DATA_BLOCK "PilzData"   // DB2702
{ S7_Optimized_Access := 'FALSE' }
// stored: AutoNumber false
   VAR RETAIN
      "85A1" : Struct
         I8 : Bool;   // Light Current 1.1
         I9 : Bool;   // Light Current 1.2
         I10 : Bool;   // Light Current 2.1
         I11 : Bool;   // Light Current 2.2
         I12 : Bool;   // Stove E Stop_2.1
         I13 : Bool;   // Stove E Stop_2.2
         I14 : Bool;   // E Stop Feedback
         I15 : Bool;   // Safety Gate Feedback
         I0 : Bool;   // Control On
         I1 : Bool;   // Control Off
         I2 : Bool;   // Spare
         I3 : Bool;   // Spare
         I4 : Bool;   // E Stop_1.1
         I5 : Bool;   // E Stop_1.2
         I6 : Bool;   // Safety Gate 1.1
         I7 : Bool;   // Safety Gate 1.2
         I24 : Bool;
         I25 : Bool;
         I26 : Bool;
         I27 : Bool;
         I28 : Bool;
         I29 : Bool;
         I30 : Bool;
         I31 : Bool;
         I16 : Bool;   // Light Current 1 feedback
         I17 : Bool;   // Light Current 2 feedback
         I18 : Bool;   // Stove E Stop feedback
         I19 : Bool;   // Spare
         I20 : Bool;   // I20
         I21 : Bool;   // I21
         I22 : Bool;   // I22
         I23 : Bool;   // I23
         O0 : Bool;
         O1 : Bool;
         O2 : Bool;
         O3 : Bool;
         Spare_1 : Bool;
         Spare_2 : Bool;
         Spare_3 : Bool;
         Spare_4 : Bool;
         Spare_5 : Bool;
         Spare_6 : Bool;
         Spare_7 : Bool;
         Spare_8 : Bool;
         Spare_9 : Bool;
         Spare_10 : Bool;
         Spare_11 : Bool;
         Spare_12 : Bool;
      END_STRUCT;
      "85A2" : Struct
         I0 : Bool;   // UnLoadingMaterialDoor 1.1
         I1 : Bool;   // UnLoadingMaterialDoor 1.2
         I2 : Bool;   // UnLoadingMaterialDoor 2.1
         I3 : Bool;   // UnLoadingMaterialDoor 2.2
         I4 : Bool;   // UnLoadingMaterialDoor 3.1
         I5 : Bool;   // UnLoadingMaterialDoor 3.2
         I6 : Bool;   // LoadingMaterialDoor 4.1
         I7 : Bool;   // LoadingMaterialDoor 4.2
         O0 : Bool;
         O1 : Bool;
         O2 : Bool;
         O3 : Bool;
         Spare_1 : Bool;
         Spare_2 : Bool;
         Spare_3 : Bool;
         Spare_4 : Bool;
      END_STRUCT;
      "85A3" : Struct
         I0 : Bool;   // MaterialDoor 1 feedback
         I1 : Bool;   // MaterialDoor 2 feedback
         I2 : Bool;   // MaterialDoor 3 feedback
         I3 : Bool;   // MaterialDoor 4 feedback
         I4 : Bool;   // Stove Door feedback 1.1
         I5 : Bool;   // Stove Door feedback 1.2
         I6 : Bool;   // Robot feedback
         I7 : Bool;   // Robot Door feedback
         O0 : Bool;
         O1 : Bool;
         O2 : Bool;
         O3 : Bool;
         Spare_1 : Bool;
         Spare_2 : Bool;
         Spare_3 : Bool;
         Spare_4 : Bool;
      END_STRUCT;
      "85A4" : Struct
         I0 : Bool;   // LoadingMaterialDoor 1.1
         I1 : Bool;   // LoadingMaterialDoor 1.2
         I2 : Bool;   // LoadingMaterialDoor 2.1
         I3 : Bool;   // LoadingMaterialDoor 2.2
         I4 : Bool;   // LoadingMaterialDoor 3.1
         I5 : Bool;   // LoadingMaterialDoor 3.2
         I6 : Bool;   // NG 2 Door 1.1
         I7 : Bool;   // NG 2 Door 1.2
         O0 : Bool;
         O1 : Bool;
         O2 : Bool;
         O3 : Bool;
         Spare_1 : Bool;
         Spare_2 : Bool;
         Spare_3 : Bool;
         Spare_4 : Bool;
      END_STRUCT;
      "85A5" : Struct
         I0 : Bool;   // Robot 1 E Stop1.1
         I1 : Bool;   // Robot 1 E Stop1.2
         I2 : Bool;   // Robot 2 E Stop1.1
         I3 : Bool;   // Robot 2 E Stop1.2
         I4 : Bool;   // Robot 3 E Stop1.1
         I5 : Bool;   // Robot 3 E Stop1.2
         I6 : Bool;   // NG 1 Door 1.1
         I7 : Bool;   // NG 1 Door 1.2
         O0 : Bool;
         O1 : Bool;
         O2 : Bool;
         O3 : Bool;
         Spare_1 : Bool;
         Spare_2 : Bool;
         Spare_3 : Bool;
         Spare_4 : Bool;
      END_STRUCT;
      TON { S7_SetPoint := 'True'} : Array[0..50] of TON_TIME;
      OK_BoxFlag : Struct
         X_Moving : Bool;
         Y_Pulling : Bool;
         X_Need_MoveBox : Bool;
         Y_Need_PullBox : Bool;
         Pushing : Bool;
         ChangeUnloadingBox : Bool;
         HMIChangeUnloadingBox : Bool;
         ManualOKBox : Bool;
         HMIManualOKBox : Int;
      END_STRUCT;
      Status : Int;
   END_VAR
BEGIN
END_DATA_BLOCK

DATA_BLOCK "GluingControl"   // DB2800
{ S7_Optimized_Access := 'FALSE' }
// stored: AutoNumber false
   VAR
      Input : Struct
         GluingDeviceReady : Bool;
         GluingFault : Bool;
         GluingRefillTank : Bool;
         GluingTankEmpty : Bool;
      END_STRUCT;
      Output : Struct
         GluingPro_X : Bool;
         GluingPro_Y : Bool;
         GluingPro_Z : Bool;
         GluingReset : Bool;
      END_STRUCT;
      Control : Struct
         Manual_X : Bool;
         Manual_Y : Bool;
         Manual_Z : Bool;
         Manual_Control : Int;
         Auto_Start : Bool;
         Auto_Y : Bool;
         Auto_Z : Bool;
         Auto_Control : Int;
         ManualTest_X : Bool;
         ManualTestStartGlue : Bool;
      END_STRUCT;
      GlueCalibratonMode : Bool;
      TON : Array[1..10] of IEC_LTIMER;
      P { S7_SetPoint := 'True'} : Array[1..10] of Bool;
      GlueInitiaStart : Bool;
   END_VAR
BEGIN
END_DATA_BLOCK

DATA_BLOCK "PalletNGData"   // DB2900
{ S7_Optimized_Access := 'FALSE' }
// stored: AutoNumber false
   VAR
      LoadingNGPallet : Struct
         NG_1_1 : Bool;
         NG_1_2 : Bool;
         NG_1_3 : Bool;
         NG_1_4 : Bool;
         NG_1_5 : Bool;
         NG_2_1 : Bool;
         NG_2_2 : Bool;
         NG_2_3 : Bool;
         NG_2_4 : Bool;
         NG_2_5 : Bool;
         NG_3_1 : Bool;
         NG_3_2 : Bool;
         NG_3_3 : Bool;
         NG_3_4 : Bool;
         NG_3_5 : Bool;
         OpenFlag : Bool;
         Status_1 : Int;
         Status_2 : Int;
         Status_3 : Int;
         Ready_1 : Bool;
         Ready_2 : Bool;
         Ready_3 : Bool;
         Ready_4 : Bool;
         Ready_5 : Bool;
         Ready_6 : Bool;
         Ready : Bool;
         Interlock_1 : Array[1..10] of Bool;
         Interlock_2 : Array[1..10] of Bool;
         Interlock_3 : Array[1..10] of Bool;
         LockStatus : Int;
      END_STRUCT;
      UnLoadingNGPallet : Struct
         NG_1_1 : Bool;
         NG_1_2 : Bool;
         NG_1_3 : Bool;
         NG_1_4 : Bool;
         NG_1_5 : Bool;
         NG_2_1 : Bool;
         NG_2_2 : Bool;
         NG_2_3 : Bool;
         NG_2_4 : Bool;
         NG_2_5 : Bool;
         NG_3_1 : Bool;
         NG_3_2 : Bool;
         NG_3_3 : Bool;
         NG_3_4 : Bool;
         NG_3_5 : Bool;
         OpenFlag : Bool;
         Status_1 : Int;
         Status_2 : Int;
         Status_3 : Int;
         Ready_1 : Bool;
         Ready_2 : Bool;
         Ready_3 : Bool;
         Ready_4 : Bool;
         Ready_5 : Bool;
         Ready_6 : Bool;
         Ready : Bool;
         Interlock_1 : Array[1..10] of Bool;
         Interlock_2 : Array[1..10] of Bool;
         Interlock_3 : Array[1..10] of Bool;
         LockStatus : Int;
      END_STRUCT;
      P : Array[0..10] of Bool;
   END_VAR
BEGIN
END_DATA_BLOCK

DATA_BLOCK "MotorControl"   // DB3100
{ S7_Optimized_Access := 'TRUE' }
// stored: AutoNumber false, MemoryReserve 100
   VAR
      Dev : Array[1..20] of "Motor_Control";
   END_VAR
BEGIN
END_DATA_BLOCK

DATA_BLOCK "MotorData"   // DB3120
{ S7_Optimized_Access := 'FALSE' }
// stored: AutoNumber false
   VAR
      Ton : Array[0..50] of TON_TIME;
      P { S7_SetPoint := 'True'} : Array[0..50] of Bool;
      "Time" : Array[0..50] of Time;
   END_VAR
BEGIN
   "Time"[0..50] := T#60s;
END_DATA_BLOCK

DATA_BLOCK "KistlerPressData1"   // DB2311
{ S7_Optimized_Access := 'FALSE' }
// stored: AutoNumber false
   VAR
      Spare : Struct
         Spare : Array[0..85] of Byte;
      END_STRUCT;
      Data : Struct
         EO01 : Struct
            "pvXMin-Y" : Real;
            "pvXMax-Y" : Real;
            "pvXMin-X" : Real;
            "pvXMax-X" : Real;
         END_STRUCT;
         EO02 : Struct
            "pvXMin-Y" : Real;
            "pvXMax-Y" : Real;
            "pvXMin-X" : Real;
            "pvXMax-X" : Real;
         END_STRUCT;
         EO03 : Struct
            "pvXMax-Y" : Real;
            "pvXMax-X" : Real;
         END_STRUCT;
      END_STRUCT;
      iWritePressData : Struct
         temp1 : Real;
      END_STRUCT;
      PressData1 : Struct
         pvBlock_X : Real;
         pvBlock_Y : Real;
      END_STRUCT;
      PressData2 : Struct
         pvBlock_X : Real;
         pvBlock_Y : Real;
      END_STRUCT;
      ManualPro : Int;
   END_VAR
BEGIN
END_DATA_BLOCK

DATA_BLOCK "KistlerPresser1_DB"   // DB2312
{ S7_Optimized_Access := 'FALSE' }
// stored: AutoNumber false
   VAR
      ShaftID : Array[0..50] of Char;
      HousingID_1 : Array[0..50] of Char;
      HousingID_2 : Array[0..50] of Char;
      Shaft : String[48];
      spare : String[48] := '46';
   END_VAR
BEGIN
END_DATA_BLOCK

DATA_BLOCK "KistlerPressData2"   // DB2321
{ S7_Optimized_Access := 'FALSE' }
// stored: AutoNumber false
   VAR
      Spare : Struct
         Spare : Array[0..85] of Byte;
      END_STRUCT;
      Data : Struct
         EO01 : Struct
            "pvXMin-Y" : Real;
            "pvXMax-Y" : Real;
            "pvXMin-X" : Real;
            "pvXMax-X" : Real;
         END_STRUCT;
         EO02 : Struct
            "pvXMin-Y" : Real;
            "pvXMax-Y" : Real;
            "pvXMin-X" : Real;
            "pvXMax-X" : Real;
         END_STRUCT;
         EO03 : Struct
            "pvXMax-Y" : Real;
            "pvXMax-X" : Real;
         END_STRUCT;
      END_STRUCT;
      iWritePressData : Struct
         temp1 : Real;
      END_STRUCT;
      PressData1 : Struct
         pvBlock_X : Real;
         pvBlock_Y : Real;
      END_STRUCT;
      ManualPro : Int;
   END_VAR
BEGIN
END_DATA_BLOCK

DATA_BLOCK "KistlerPresser2_DB"   // DB2322
{ S7_Optimized_Access := 'FALSE' }
// stored: AutoNumber false
   VAR
      ShaftID : Array[0..50] of Char;
      HousingID_1 : Array[0..50] of Char;
      HousingID_2 : Array[0..50] of Char;
      Shaft : String[48];
      spare : String[48] := '46';
   END_VAR
BEGIN
END_DATA_BLOCK

DATA_BLOCK "ST10_FB_Tower_4Lamp_DB"
{ S7_Optimized_Access := 'TRUE' }
VERSION : 0.1
NON_RETAIN
// ATTRIBUTES
// AUTO_NUMBER = False
// BLOCK_NUMBER = 5050
// END_ATTRIBUTES
"FB_Tower_4Lamp"

BEGIN

END_DATA_BLOCK

DATA_BLOCK "DB_ProcessSlots"
{ S7_Optimized_Access := 'TRUE' }
VERSION : 0.1
// ATTRIBUTES
// AUTO_NUMBER = False
// BLOCK_NUMBER = 2600
// END_ATTRIBUTES
   VAR 
      Slots : Array[1..16] of "UDT_ProcessSlot";
   END_VAR


BEGIN
   Slots[1].SlotID := 1;
   Slots[1].PositionTag := 'A_ScanRotate';
   Slots[2].SlotID := 2;
   Slots[2].PositionTag := 'F_Robot1Grip1';
   Slots[3].SlotID := 3;
   Slots[3].PositionTag := 'F_Robot1Grip2';
   Slots[4].SlotID := 4;
   Slots[4].PositionTag := 'B_Press1';
   Slots[5].SlotID := 5;
   Slots[5].PositionTag := 'C_Glue';
   Slots[6].SlotID := 6;
   Slots[6].PositionTag := 'F_Robot2Grip1';
   Slots[7].SlotID := 7;
   Slots[7].PositionTag := 'F_Robot2Grip2';
   Slots[8].SlotID := 8;
   Slots[8].PositionTag := 'C_GlueNGBuffer';
   Slots[9].SlotID := 9;
   Slots[9].PositionTag := 'C_MagnScanNGBuffer';
   Slots[10].SlotID := 10;
   Slots[10].PositionTag := 'B_Press2';
   Slots[11].SlotID := 11;
   Slots[11].PositionTag := 'F_Robot3Grip1';
   Slots[12].SlotID := 12;
   Slots[12].PositionTag := 'F_Robot3Grip2';
   Slots[13].SlotID := 13;
   Slots[13].PositionTag := 'H_ShafeLine';
   Slots[14].SlotID := 14;
   Slots[14].PositionTag := 'J_ShafeLine';
   Slots[15].SlotID := 15;
   Slots[15].PositionTag := 'K_ShafeLine';
   Slots[16].SlotID := 16;
   Slots[16].PositionTag := 'L_ShafeLine';

END_DATA_BLOCK

DATA_BLOCK "DB_ProcessSlots_Global"
{ S7_Optimized_Access := 'TRUE' }
VERSION : 0.1
// ATTRIBUTES
// AUTO_NUMBER = False
// BLOCK_NUMBER = 2601
// END_ATTRIBUTES
   VAR 
      SlotHasProduct : Array[1..16] of Bool;
      SlotLocked : Array[1..16] of Bool;
      SlotPendingWrite : Array[1..16] of Bool;
      ActiveRecipeID : Int;
      ActiveRecipeVersion : String[18];
      BufferIndex : Int;
   END_VAR


BEGIN
   ActiveRecipeID := 1;
   ActiveRecipeVersion := 'INIT';
   BufferIndex := 1;

END_DATA_BLOCK

DATA_BLOCK "DB_RecipeActiveNew"
{ S7_Optimized_Access := 'TRUE' }
VERSION : 0.1
// ATTRIBUTES
// AUTO_NUMBER = False
// BLOCK_NUMBER = 2701
// END_ATTRIBUTES
   VAR 
      Header : "UDT_RecipeHeader";
      SubProcess : Array[1..16] of "UDT_SubProcessRecipe";
      FixtureCodes : Array[1..16] of String[128];
      GripperCodes : Array[1..12] of String[128];
      PressPrograms : Array[1..4] of Int;
      VisionPrograms : Array[1..8] of Int;
   END_VAR


BEGIN
   Header.ProductName := 'ACTIVE';
   Header.ProductID := 'ACTIVE';
   Header.RecipeVersion := 'PENDING';
   Header.Enabled := FALSE;

END_DATA_BLOCK

DATA_BLOCK "DB_RecipeMaster"
{ S7_Optimized_Access := 'TRUE' }
VERSION : 0.1
// ATTRIBUTES
// AUTO_NUMBER = False
// BLOCK_NUMBER = 2700
// END_ATTRIBUTES
   VAR 
      Header : "UDT_RecipeHeader";
      SubProcess : Array[1..32] of "UDT_SubProcessRecipe";
      FixtureCodes : Array[1..16] of String[128];
      GripperCodes : Array[1..18] of String[128];
      VisionPrograms : Array[1..16] of Int;
   END_VAR


BEGIN
   Header.ProductName := 'Product_1';
   Header.ProductID := 'P1';
   Header.RecipeVersion := 'V1.0';
   Header.FixtureFamily := 1;
   Header.Enabled := TRUE;
   Header.CreatedBy := 'OP10';
   Header.UpdatedBy := 'OP10';
   Header.Comment := 'Seed recipe migrated from ST10_RecipeDB';

   FixtureCodes[1] := 'SZ23055-OP010-E-Compressor-ring1 Loading tooling-1';
   FixtureCodes[2] := 'SZ23055-OP010-E-Compressor-ring1 Loading tooling-2';
   FixtureCodes[3] := 'SZ23055-OP010-E-Compressor-ring1 Loading tooling-3';
   FixtureCodes[4] := 'SZ23055-OP010-E-Compressor-ring1 Loading tooling-4';
   FixtureCodes[5] := 'SZ23055-OP010-E-Compressor-ring1 Loading tooling-5';
   FixtureCodes[6] := 'SZ23055-OP010-E-Compressor-ring1 Loading tooling-6';
   FixtureCodes[7] := 'SZ23055-OP010-E-Compressor-ring1 Loading tooling-7';
   FixtureCodes[8] := 'SZ23055-OP010-E-Compressor-ring1 Loading tooling-8';
   FixtureCodes[9] := 'SZ23055-OP010-E-Compressor-ring2 Loading tooling-1';
   FixtureCodes[10] := 'SZ23055-OP010-E-Compressor-ring2 Loading tooling-2';
   FixtureCodes[11] := 'SZ23055-OP010-E-Compressor-ring2 Loading tooling-3';
   FixtureCodes[12] := 'SZ23055-OP010-E-Compressor-ring2 Loading tooling-4';

   GripperCodes[1] := 'SZ23055-OP010-E-Compressor-robot1 ring1 Left clamping jaw tooling-1';
   GripperCodes[2] := 'SZ23055-OP010-E-Compressor-robot1 ring1 Right clamping jaw tooling-2';
   GripperCodes[3] := 'SZ23055-OP010-E-Compressor-robot1 shaft Left clamping jaw tooling-1';
   GripperCodes[4] := 'SZ23055-OP010-E-Compressor-robot1 shaft Right clamping jaw tooling-2';
   GripperCodes[5] := 'SZ23055-OP010-E-Compressor-robot2 shaft Right clamping jaw tooling-2';
   GripperCodes[6] := 'SZ23055-OP010-E-Compressor-robot2 shaft Left clamping jaw tooling-1';

END_DATA_BLOCK

DATA_BLOCK "ST10_CountCycleTimeMain_DB"
{ S7_Optimized_Access := 'TRUE' }
VERSION : 0.1
NON_RETAIN
// ATTRIBUTES
// AUTO_NUMBER = False
// BLOCK_NUMBER = 1009
// END_ATTRIBUTES
"ST10_CountCycleTimeMain"

BEGIN

END_DATA_BLOCK

DATA_BLOCK "DB_MESLoadData"
{ S7_Optimized_Access := 'TRUE' }
VERSION : 0.1
// ATTRIBUTES
// AUTO_NUMBER = False
// BLOCK_NUMBER = 2800
// END_ATTRIBUTES
   VAR 
      Station1 : "UDT_MESLoadData";
      Station2 : "UDT_MESLoadData";
      Station3 : "UDT_MESLoadData";
      Station4 : "UDT_MESLoadData";
   END_VAR


BEGIN

END_DATA_BLOCK

DATA_BLOCK "DT-Chars_DB"
{ S7_Optimized_Access := 'FALSE' }
VERSION : 0.1
NON_RETAIN
// ATTRIBUTES
// AUTO_NUMBER = False
// BLOCK_NUMBER = 2360
// END_ATTRIBUTES
"DT-Chars"

BEGIN

END_DATA_BLOCK

DATA_BLOCK "MES_CHeck_DB"
{ S7_Optimized_Access := 'TRUE' }
VERSION : 0.1
NON_RETAIN
// ATTRIBUTES
// AUTO_NUMBER = False
// BLOCK_NUMBER = 111
// END_ATTRIBUTES
"MES_CHeck"

BEGIN

END_DATA_BLOCK

DATA_BLOCK "PartDataManage_Part1_DB"
{ S7_Optimized_Access := 'TRUE' }
VERSION : 0.1
NON_RETAIN
// ATTRIBUTES
// AUTO_NUMBER = True
// BLOCK_NUMBER = 1501
// END_ATTRIBUTES
"PartDataManage"

BEGIN

END_DATA_BLOCK

DATA_BLOCK "PartDataManage_Part2_DB"
{ S7_Optimized_Access := 'TRUE' }
VERSION : 0.1
NON_RETAIN
"PartDataManage"

BEGIN

END_DATA_BLOCK

DATA_BLOCK "PartDataManage_Part3_DB"
{ S7_Optimized_Access := 'TRUE' }
VERSION : 0.1
NON_RETAIN
// ATTRIBUTES
// AUTO_NUMBER = True
// BLOCK_NUMBER = 1503
// END_ATTRIBUTES
"PartDataManage"

BEGIN

END_DATA_BLOCK

DATA_BLOCK "PartDataManage_Part4_DB"
{ S7_Optimized_Access := 'TRUE' }
VERSION : 0.1
NON_RETAIN
// ATTRIBUTES
// AUTO_NUMBER = True
// BLOCK_NUMBER = 1504
// END_ATTRIBUTES
"PartDataManage"

BEGIN

END_DATA_BLOCK

DATA_BLOCK "MB_CLIENT_DB"
{InstructionName := 'MB_CLIENT';
 LibVersion := '5.1';
 S7_Optimized_Access := 'TRUE' }
AUTHOR : SIMATIC
FAMILY : MBUS_TCP
NAME : MB_CLI
VERSION : 5.1
NON_RETAIN
MB_CLIENT

BEGIN

END_DATA_BLOCK

DATA_BLOCK "ST10_SystemModeFB_iDB"
{ S7_Optimized_Access := 'TRUE' }
VERSION : 0.1
NON_RETAIN
// ATTRIBUTES
// AUTO_NUMBER = False
// BLOCK_NUMBER = 1000
// END_ATTRIBUTES
"SystemMode"

BEGIN

END_DATA_BLOCK

DATA_BLOCK "AutoProcessDataPopUp_DB"
{ S7_Optimized_Access := 'TRUE' }
VERSION : 0.1
NON_RETAIN
// ATTRIBUTES
// AUTO_NUMBER = True
// BLOCK_NUMBER = 2
// END_ATTRIBUTES
"AutoProcessDataPopUp"

BEGIN

END_DATA_BLOCK

DATA_BLOCK "ST10_Flow11_A2TableScan_iDB"
{ S7_Optimized_Access := 'TRUE' }
VERSION : 0.1
NON_RETAIN
// ATTRIBUTES
// AUTO_NUMBER = False
// BLOCK_NUMBER = 1081
// END_ATTRIBUTES
"ST10_Flow11_A2TableScan"

BEGIN

END_DATA_BLOCK

DATA_BLOCK "ST10_Flow12_A2TableUnloading_iDB"
{ S7_Optimized_Access := 'TRUE' }
VERSION : 0.1
NON_RETAIN
// ATTRIBUTES
// AUTO_NUMBER = False
// BLOCK_NUMBER = 1082
// END_ATTRIBUTES
"ST10_Flow12_A2TableUnloading"

BEGIN

END_DATA_BLOCK

DATA_BLOCK "ST10_Flow14_B2Press_iDB"
{ S7_Optimized_Access := 'TRUE' }
VERSION : 0.1
NON_RETAIN
// ATTRIBUTES
// AUTO_NUMBER = False
// BLOCK_NUMBER = 1084
// END_ATTRIBUTES
"ST10_Flow14_B2Press"

BEGIN

END_DATA_BLOCK

DATA_BLOCK "ST10_Flow15_FRobot_3_iDB"
{ S7_Optimized_Access := 'TRUE' }
VERSION : 0.1
NON_RETAIN
// ATTRIBUTES
// AUTO_NUMBER = False
// BLOCK_NUMBER = 1085
// END_ATTRIBUTES
"ST10_Flow15_FRobot_3"

BEGIN

END_DATA_BLOCK

DATA_BLOCK "ST10_Flow1_A1TableScan_iDB"
{ S7_Optimized_Access := 'TRUE' }
VERSION : 0.1
NON_RETAIN
"ST10_Flow1_A1TableScan"

BEGIN

END_DATA_BLOCK

DATA_BLOCK "ST10_Flow21_HShaftLifting_iDB"
{ S7_Optimized_Access := 'TRUE' }
VERSION : 0.1
NON_RETAIN
// ATTRIBUTES
// AUTO_NUMBER = False
// BLOCK_NUMBER = 1091
// END_ATTRIBUTES
"ST10_Flow21_HShaftLifting"

BEGIN

END_DATA_BLOCK

DATA_BLOCK "ST10_Flow22_JMagnetLifting_iDB"
{ S7_Optimized_Access := 'TRUE' }
VERSION : 0.1
NON_RETAIN
"ST10_Flow22_JMagnetLifting"

BEGIN

END_DATA_BLOCK

DATA_BLOCK "ST10_Flow23_KReserveLifting_iDB"
{ S7_Optimized_Access := 'TRUE' }
VERSION : 0.1
NON_RETAIN
// ATTRIBUTES
// AUTO_NUMBER = False
// BLOCK_NUMBER = 1093
// END_ATTRIBUTES
"ST10_Flow23_KReserveLifting"

BEGIN

END_DATA_BLOCK

DATA_BLOCK "ST10_Flow24_LUnloadingTrans_iDB"
{ S7_Optimized_Access := 'TRUE' }
VERSION : 0.1
NON_RETAIN
// ATTRIBUTES
// AUTO_NUMBER = False
// BLOCK_NUMBER = 1094
// END_ATTRIBUTES
"ST10_Flow24_LUnloadingTrans"

BEGIN

END_DATA_BLOCK

DATA_BLOCK "ST10_Flow25_HShaftLoad&Unload_iDB"
{ S7_Optimized_Access := 'TRUE' }
VERSION : 0.1
NON_RETAIN
// ATTRIBUTES
// AUTO_NUMBER = False
// BLOCK_NUMBER = 1095
// END_ATTRIBUTES
"ST10_Flow25_HShaftLoad&Unload"

BEGIN

END_DATA_BLOCK

DATA_BLOCK "ST10_Flow26_JMagnetLoad&Unload_iDB"
{ S7_Optimized_Access := 'TRUE' }
VERSION : 0.1
NON_RETAIN
// ATTRIBUTES
// AUTO_NUMBER = False
// BLOCK_NUMBER = 1096
// END_ATTRIBUTES
"ST10_Flow26_JMagnetLoad&Unload"

BEGIN

END_DATA_BLOCK

DATA_BLOCK "ST10_Flow27_KReserveLoad&Unload_iDB"
{ S7_Optimized_Access := 'TRUE' }
VERSION : 0.1
NON_RETAIN
// ATTRIBUTES
// AUTO_NUMBER = False
// BLOCK_NUMBER = 1097
// END_ATTRIBUTES
"ST10_Flow27_KReserveLoad&Unload"

BEGIN

END_DATA_BLOCK

DATA_BLOCK "ST10_Flow28_LUnloadingLoad&Unload_IiDB"
{ S7_Optimized_Access := 'TRUE' }
VERSION : 0.1
NON_RETAIN
"ST10_Flow28_LUnloadingLoad&Unload"

BEGIN

END_DATA_BLOCK

DATA_BLOCK "ST10_Flow2_A1TableUnloading_iDB"
{ S7_Optimized_Access := 'TRUE' }
VERSION : 0.1
NON_RETAIN
"ST10_Flow2_A1TableUnloading"

BEGIN

END_DATA_BLOCK

DATA_BLOCK "ST10_Flow3_A1RotaryScan_iDB"
{ S7_Optimized_Access := 'TRUE' }
VERSION : 0.1
NON_RETAIN
// ATTRIBUTES
// AUTO_NUMBER = False
// BLOCK_NUMBER = 1073
// END_ATTRIBUTES
"ST10_Flow3_A1RotaryShaftScan"

BEGIN

END_DATA_BLOCK

DATA_BLOCK "ST10_Flow4_B1Press_iDB"
{ S7_Optimized_Access := 'TRUE' }
VERSION : 0.1
NON_RETAIN
"ST10_Flow4_B1Press"

BEGIN

END_DATA_BLOCK

DATA_BLOCK "ST10_Flow5_FRobot_1_iDB"
{ S7_Optimized_Access := 'TRUE' }
VERSION : 0.1
NON_RETAIN
"ST10_Flow5_FRobot_1"

BEGIN

END_DATA_BLOCK

DATA_BLOCK "ST10_Flow6_FixtureCodeScan_iDB"
{ S7_Optimized_Access := 'TRUE' }
VERSION : 0.1
NON_RETAIN
"ST10_Flow6_ToolCodeScan"

BEGIN

END_DATA_BLOCK

DATA_BLOCK "ST10_Flow7_CGlueing_iDB"
{ S7_Optimized_Access := 'TRUE' }
VERSION : 0.1
NON_RETAIN
"ST10_Flow7_CGlueing"

BEGIN

END_DATA_BLOCK

DATA_BLOCK "ST10_Flow8_FRobot_2_iDB"
{ S7_Optimized_Access := 'TRUE' }
VERSION : 0.1
NON_RETAIN
// ATTRIBUTES
// AUTO_NUMBER = False
// BLOCK_NUMBER = 1078
// END_ATTRIBUTES
"ST10_Flow8_FRobot_2"

BEGIN

END_DATA_BLOCK

DATA_BLOCK "ST10_MaterialGate1_DB"
{ S7_Optimized_Access := 'FALSE' }
VERSION : 0.1
NON_RETAIN
// ATTRIBUTES
// AUTO_NUMBER = False
// BLOCK_NUMBER = 1151
// END_ATTRIBUTES
"SafetyGate"

BEGIN

END_DATA_BLOCK

DATA_BLOCK "ST10_MaterialGate2_DB"
{ S7_Optimized_Access := 'FALSE' }
VERSION : 0.1
NON_RETAIN
// ATTRIBUTES
// AUTO_NUMBER = False
// BLOCK_NUMBER = 1152
// END_ATTRIBUTES
"SafetyGate"

BEGIN

END_DATA_BLOCK

DATA_BLOCK "ST10_MaterialGate3_DB"
{ S7_Optimized_Access := 'FALSE' }
VERSION : 0.1
NON_RETAIN
// ATTRIBUTES
// AUTO_NUMBER = False
// BLOCK_NUMBER = 1153
// END_ATTRIBUTES
"SafetyGate"

BEGIN

END_DATA_BLOCK

DATA_BLOCK "ST10_MaterialGate4_DB"
{ S7_Optimized_Access := 'FALSE' }
VERSION : 0.1
NON_RETAIN
// ATTRIBUTES
// AUTO_NUMBER = False
// BLOCK_NUMBER = 1154
// END_ATTRIBUTES
"SafetyGate"

BEGIN

END_DATA_BLOCK

DATA_BLOCK "ST10_MaterialGate5_DB"
{ S7_Optimized_Access := 'FALSE' }
VERSION : 0.1
NON_RETAIN
// ATTRIBUTES
// AUTO_NUMBER = False
// BLOCK_NUMBER = 1155
// END_ATTRIBUTES
"SafetyGate"

BEGIN

END_DATA_BLOCK

DATA_BLOCK "ST10_MaterialGate6_DB"
{ S7_Optimized_Access := 'FALSE' }
VERSION : 0.1
NON_RETAIN
// ATTRIBUTES
// AUTO_NUMBER = False
// BLOCK_NUMBER = 1156
// END_ATTRIBUTES
"SafetyGate"

BEGIN

END_DATA_BLOCK

DATA_BLOCK "ST10_MaterialGate7_DB"
{ S7_Optimized_Access := 'FALSE' }
VERSION : 0.1
NON_RETAIN
// ATTRIBUTES
// AUTO_NUMBER = False
// BLOCK_NUMBER = 1157
// END_ATTRIBUTES
"SafetyGate"

BEGIN

END_DATA_BLOCK

DATA_BLOCK "ST10_NGGate1_DB"
{ S7_Optimized_Access := 'FALSE' }
VERSION : 0.1
NON_RETAIN
// ATTRIBUTES
// AUTO_NUMBER = False
// BLOCK_NUMBER = 1158
// END_ATTRIBUTES
"SafetyGate"

BEGIN

END_DATA_BLOCK

DATA_BLOCK "ST10_NGGate2_DB"
{ S7_Optimized_Access := 'FALSE' }
VERSION : 0.1
NON_RETAIN
// ATTRIBUTES
// AUTO_NUMBER = False
// BLOCK_NUMBER = 1159
// END_ATTRIBUTES
"SafetyGate"

BEGIN

END_DATA_BLOCK

DATA_BLOCK "ST10_SafetyGate1_DB"
{ S7_Optimized_Access := 'FALSE' }
VERSION : 0.1
NON_RETAIN
// ATTRIBUTES
// AUTO_NUMBER = False
// BLOCK_NUMBER = 1141
// END_ATTRIBUTES
"SafetyGate"

BEGIN

END_DATA_BLOCK

DATA_BLOCK "ST10_SafetyGate2_DB"
{ S7_Optimized_Access := 'FALSE' }
VERSION : 0.1
NON_RETAIN
// ATTRIBUTES
// AUTO_NUMBER = False
// BLOCK_NUMBER = 1142
// END_ATTRIBUTES
"SafetyGate"

BEGIN

END_DATA_BLOCK

DATA_BLOCK "ST10_SafetyGate3_DB"
{ S7_Optimized_Access := 'FALSE' }
VERSION : 0.1
NON_RETAIN
// ATTRIBUTES
// AUTO_NUMBER = False
// BLOCK_NUMBER = 1143
// END_ATTRIBUTES
"SafetyGate"

BEGIN

END_DATA_BLOCK

DATA_BLOCK "ST10_SafetyGate4_DB"
{ S7_Optimized_Access := 'FALSE' }
VERSION : 0.1
NON_RETAIN
// ATTRIBUTES
// AUTO_NUMBER = False
// BLOCK_NUMBER = 1144
// END_ATTRIBUTES
"SafetyGate"

BEGIN

END_DATA_BLOCK

DATA_BLOCK "ST10_SafetyGate5_DB"
{ S7_Optimized_Access := 'FALSE' }
VERSION : 0.1
NON_RETAIN
// ATTRIBUTES
// AUTO_NUMBER = False
// BLOCK_NUMBER = 1145
// END_ATTRIBUTES
"SafetyGate"

BEGIN

END_DATA_BLOCK

DATA_BLOCK "ST10_SafetyGate6_DB"
{ S7_Optimized_Access := 'FALSE' }
VERSION : 0.1
NON_RETAIN
"SafetyGate"

BEGIN

END_DATA_BLOCK

DATA_BLOCK "ST10_SafetyGate7_DB"
{ S7_Optimized_Access := 'FALSE' }
VERSION : 0.1
NON_RETAIN
"SafetyGate"

BEGIN

END_DATA_BLOCK

DATA_BLOCK "ST10_SafetyGate8_DB"
{ S7_Optimized_Access := 'FALSE' }
VERSION : 0.1
NON_RETAIN
// ATTRIBUTES
// AUTO_NUMBER = False
// BLOCK_NUMBER = 1148
// END_ATTRIBUTES
"SafetyGate"

BEGIN

END_DATA_BLOCK

DATA_BLOCK "ST10_SafetyGate9_DB"
{ S7_Optimized_Access := 'FALSE' }
VERSION : 0.1
NON_RETAIN
// ATTRIBUTES
// AUTO_NUMBER = False
// BLOCK_NUMBER = 1149
// END_ATTRIBUTES
"SafetyGate"

BEGIN

END_DATA_BLOCK

DATA_BLOCK "ST10_Stopper_FB_DB"
{ S7_Optimized_Access := 'TRUE' }
VERSION : 0.1
NON_RETAIN
// ATTRIBUTES
// AUTO_NUMBER = False
// BLOCK_NUMBER = 1160
// END_ATTRIBUTES
"ST10_Stopper_FB"

BEGIN

END_DATA_BLOCK

DATA_BLOCK "KeyenceSR1000Ctrl_800A1DB"
{ S7_Optimized_Access := 'FALSE' }
VERSION : 0.1
NON_RETAIN
"KeyenceSR1000Ctrl"

BEGIN

END_DATA_BLOCK

DATA_BLOCK "KeyenceSR1000Ctrl_801A1DB"
{ S7_Optimized_Access := 'FALSE' }
VERSION : 0.1
NON_RETAIN
// ATTRIBUTES
// AUTO_NUMBER = False
// BLOCK_NUMBER = 1801
// END_ATTRIBUTES
"KeyenceSR1000Ctrl"

BEGIN

END_DATA_BLOCK

DATA_BLOCK "KeyenceSR1000Ctrl_802A1DB"
{ S7_Optimized_Access := 'FALSE' }
VERSION : 0.1
NON_RETAIN
// ATTRIBUTES
// AUTO_NUMBER = False
// BLOCK_NUMBER = 1806
// END_ATTRIBUTES
"KeyenceSR1000Ctrl"

BEGIN

END_DATA_BLOCK

DATA_BLOCK "KeyenceSR1000Ctrl_803A1DB"
{ S7_Optimized_Access := 'FALSE' }
VERSION : 0.1
NON_RETAIN
// ATTRIBUTES
// AUTO_NUMBER = False
// BLOCK_NUMBER = 1802
// END_ATTRIBUTES
"KeyenceSR1000Ctrl"

BEGIN

END_DATA_BLOCK

DATA_BLOCK "KeyenceSR1000Ctrl_804A1DB"
{ S7_Optimized_Access := 'FALSE' }
VERSION : 0.1
NON_RETAIN
// ATTRIBUTES
// AUTO_NUMBER = False
// BLOCK_NUMBER = 1803
// END_ATTRIBUTES
"KeyenceSR1000Ctrl"

BEGIN

END_DATA_BLOCK

DATA_BLOCK "KeyenceSR1000Ctrl_805A1DB"
{ S7_Optimized_Access := 'FALSE' }
VERSION : 0.1
NON_RETAIN
// ATTRIBUTES
// AUTO_NUMBER = False
// BLOCK_NUMBER = 1807
// END_ATTRIBUTES
"KeyenceSR1000Ctrl"

BEGIN

END_DATA_BLOCK

DATA_BLOCK "KeyenceSR1000Ctrl_806A1DB"
{ S7_Optimized_Access := 'FALSE' }
VERSION : 0.1
NON_RETAIN
// ATTRIBUTES
// AUTO_NUMBER = False
// BLOCK_NUMBER = 1804
// END_ATTRIBUTES
"KeyenceSR1000Ctrl"

BEGIN

END_DATA_BLOCK

DATA_BLOCK "KeyenceSR1000Ctrl_807A1DB"
{ S7_Optimized_Access := 'FALSE' }
VERSION : 0.1
NON_RETAIN
// ATTRIBUTES
// AUTO_NUMBER = False
// BLOCK_NUMBER = 1808
// END_ATTRIBUTES
"KeyenceSR1000Ctrl"

BEGIN

END_DATA_BLOCK

DATA_BLOCK "Call_KeyenceCheckerIV_DB"
{ S7_Optimized_Access := 'TRUE' }
VERSION : 0.1
NON_RETAIN
"Call_KeyenceCheckerIV"

BEGIN

END_DATA_BLOCK

DATA_BLOCK "Axis_FB_DB"
{ S7_Optimized_Access := 'FALSE' }
VERSION : 0.1
// ATTRIBUTES
// AUTO_NUMBER = False
// BLOCK_NUMBER = 2200
// END_ATTRIBUTES
"Axis_FB"

BEGIN

END_DATA_BLOCK

DATA_BLOCK "IAI_Position_DB"
{ S7_Optimized_Access := 'TRUE' }
VERSION : 0.1
NON_RETAIN
"IAI_Position"

BEGIN

END_DATA_BLOCK

DATA_BLOCK "KukaRobot1_CtrlDB"
{ S7_Optimized_Access := 'FALSE' }
VERSION : 0.1
// ATTRIBUTES
// AUTO_NUMBER = False
// BLOCK_NUMBER = 2401
// END_ATTRIBUTES
"KukaRobot1_Ctrl"

BEGIN

END_DATA_BLOCK

DATA_BLOCK "KukaRobot2_CtrlDB"
{ S7_Optimized_Access := 'FALSE' }
VERSION : 0.1
// ATTRIBUTES
// AUTO_NUMBER = False
// BLOCK_NUMBER = 2402
// END_ATTRIBUTES
"KukaRobot2_Ctrl"

BEGIN

END_DATA_BLOCK

DATA_BLOCK "KukaRobot3_CtrlDB"
{ S7_Optimized_Access := 'FALSE' }
VERSION : 0.1
// ATTRIBUTES
// AUTO_NUMBER = False
// BLOCK_NUMBER = 2403
// END_ATTRIBUTES
"KukaRobot3_Ctrl"

BEGIN

END_DATA_BLOCK

DATA_BLOCK "V90Servo_DB"
{ S7_Optimized_Access := 'TRUE' }
VERSION : 0.1
NON_RETAIN
"V90_Servo"

BEGIN

END_DATA_BLOCK

DATA_BLOCK "ST10_StopperCtrl_DB"
{ S7_Optimized_Access := 'FALSE' }
VERSION : 0.1
NON_RETAIN
// ATTRIBUTES
// AUTO_NUMBER = False
// BLOCK_NUMBER = 2601
// END_ATTRIBUTES
"ST10_StopperCtrl"

BEGIN

END_DATA_BLOCK

DATA_BLOCK "PilzData_fb_DB"
{ S7_Optimized_Access := 'TRUE' }
VERSION : 0.1
NON_RETAIN
"PilzData_fb"

BEGIN

END_DATA_BLOCK

DATA_BLOCK "Pilz_fb_DB"
{ S7_Optimized_Access := 'FALSE' }
VERSION : 0.1
NON_RETAIN
// ATTRIBUTES
// AUTO_NUMBER = False
// BLOCK_NUMBER = 2700
// END_ATTRIBUTES
"Pilz_fb"

BEGIN

END_DATA_BLOCK

DATA_BLOCK "NG_DB"
{ S7_Optimized_Access := 'TRUE' }
VERSION : 0.1
NON_RETAIN
"NG"

BEGIN

END_DATA_BLOCK

DATA_BLOCK "MotorContro_DB_1"
{ S7_Optimized_Access := 'TRUE' }
VERSION : 0.1
NON_RETAIN
"MotorContro"

BEGIN

END_DATA_BLOCK

DATA_BLOCK "MotorContro_DB_11"
{ S7_Optimized_Access := 'TRUE' }
VERSION : 0.1
NON_RETAIN
// ATTRIBUTES
// AUTO_NUMBER = False
// BLOCK_NUMBER = 3111
// END_ATTRIBUTES
"MotorContro"

BEGIN

END_DATA_BLOCK

DATA_BLOCK "MotorContro_DB_12"
{ S7_Optimized_Access := 'TRUE' }
VERSION : 0.1
NON_RETAIN
// ATTRIBUTES
// AUTO_NUMBER = False
// BLOCK_NUMBER = 3112
// END_ATTRIBUTES
"MotorContro"

BEGIN

END_DATA_BLOCK

DATA_BLOCK "MotorContro_DB_13"
{ S7_Optimized_Access := 'TRUE' }
VERSION : 0.1
NON_RETAIN
// ATTRIBUTES
// AUTO_NUMBER = False
// BLOCK_NUMBER = 3113
// END_ATTRIBUTES
"MotorContro"

BEGIN

END_DATA_BLOCK

DATA_BLOCK "MotorContro_DB_14"
{ S7_Optimized_Access := 'TRUE' }
VERSION : 0.1
NON_RETAIN
// ATTRIBUTES
// AUTO_NUMBER = False
// BLOCK_NUMBER = 3114
// END_ATTRIBUTES
"MotorContro"

BEGIN

END_DATA_BLOCK

DATA_BLOCK "MotorContro_DB_15"
{ S7_Optimized_Access := 'TRUE' }
VERSION : 0.1
NON_RETAIN
// ATTRIBUTES
// AUTO_NUMBER = False
// BLOCK_NUMBER = 3115
// END_ATTRIBUTES
"MotorContro"

BEGIN

END_DATA_BLOCK

DATA_BLOCK "MotorContro_DB_16"
{ S7_Optimized_Access := 'TRUE' }
VERSION : 0.1
NON_RETAIN
// ATTRIBUTES
// AUTO_NUMBER = False
// BLOCK_NUMBER = 3116
// END_ATTRIBUTES
"MotorContro"

BEGIN

END_DATA_BLOCK

DATA_BLOCK "MotorContro_DB_17"
{ S7_Optimized_Access := 'TRUE' }
VERSION : 0.1
NON_RETAIN
// ATTRIBUTES
// AUTO_NUMBER = False
// BLOCK_NUMBER = 3117
// END_ATTRIBUTES
"MotorContro"

BEGIN

END_DATA_BLOCK

DATA_BLOCK "MotorContro_DB_2"
{ S7_Optimized_Access := 'TRUE' }
VERSION : 0.1
NON_RETAIN
"MotorContro"

BEGIN

END_DATA_BLOCK

DATA_BLOCK "MotorContro_DB_3"
{ S7_Optimized_Access := 'TRUE' }
VERSION : 0.1
NON_RETAIN
// ATTRIBUTES
// AUTO_NUMBER = False
// BLOCK_NUMBER = 3103
// END_ATTRIBUTES
"MotorContro"

BEGIN

END_DATA_BLOCK

DATA_BLOCK "MotorContro_DB_4"
{ S7_Optimized_Access := 'TRUE' }
VERSION : 0.1
NON_RETAIN
"MotorContro"

BEGIN

END_DATA_BLOCK

DATA_BLOCK "ST10_FB_S7connect_IDB"
{ S7_Optimized_Access := 'TRUE' }
VERSION : 0.1
NON_RETAIN
// ATTRIBUTES
// AUTO_NUMBER = False
// BLOCK_NUMBER = 900
// END_ATTRIBUTES
"ST10_FB_S7connect"

BEGIN

END_DATA_BLOCK

DATA_BLOCK "DB_maXYmosNC1"
{ S7_Optimized_Access := 'FALSE' }
VERSION : 0.1
NON_RETAIN
// ATTRIBUTES
// AUTO_NUMBER = False
// BLOCK_NUMBER = 2310
// END_ATTRIBUTES
"KistlerPresser _FB"

BEGIN

END_DATA_BLOCK

DATA_BLOCK "DB_maXYmosNC2"
{ S7_Optimized_Access := 'FALSE' }
VERSION : 0.1
NON_RETAIN
// ATTRIBUTES
// AUTO_NUMBER = False
// BLOCK_NUMBER = 2320
// END_ATTRIBUTES
"KistlerPresser _FB"

BEGIN

END_DATA_BLOCK

ORGANIZATION_BLOCK "01_OB1"   // OB1, LAD, ProgramCycle
TITLE = "Main Program Sweep (Cycle)"
{ S7_Optimized_Access := 'FALSE' }
AUTHOR : STD
FAMILY : System
VERSION : 2.0
// 系统程序段无需改动
// stored: AutoNumber false, SetENOAutomatically false
   VAR_TEMP
      OB1_EV_CLASS : Byte;   // Bits 0-3 = 1 (Coming event), Bits 4-7 = 1 (Event class 1)
      OB1_SCAN_1 : Byte;   // 1 (Cold restart scan 1 of OB 1), 3 (Scan 2-n of OB 1)
      OB1_PRIORITY : Byte;   // Priority of OB Execution
      OB1_OB_NUMBR : Byte;   // 1 (Organization block 1, OB1)
      OB1_RESERVED_1 : Byte;   // Reserved for system
      OB1_RESERVED_2 : Byte;   // Reserved for system
      OB1_PREV_CYCLE : Int;   // Cycle time of previous OB1 scan (milliseconds)
      OB1_MIN_CYCLE : Int;   // Minimum cycle time of OB1 (milliseconds)
      OB1_MAX_CYCLE : Int;   // Maximum cycle time of OB1 (milliseconds)
      OB1_DATE_TIME : Date_And_Time;   // Date and time OB1 started
      i : Int;
   END_VAR
   VAR_TEMP   // added for the SCL form of the ladder/FBD networks
      _w1 : Bool;
   END_VAR
BEGIN

REGION Network 1: Normal ON & OFF
   // 系统程序段
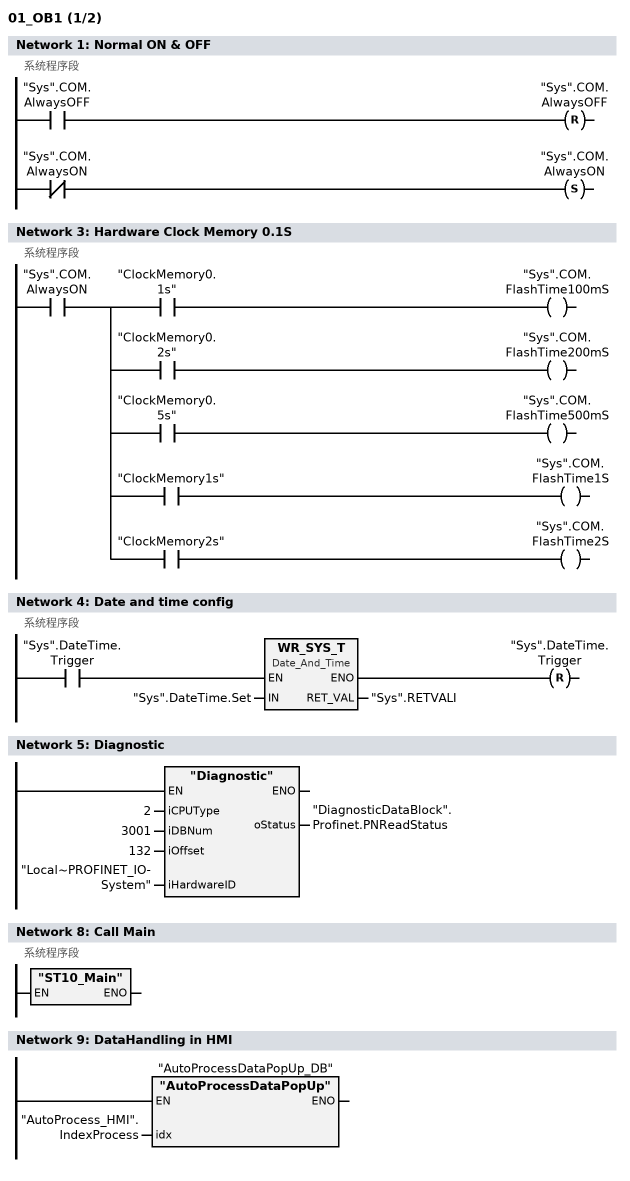
   RUNG wire#powerrail
      Contact( "Sys".COM.AlwaysOFF )
      R_Coil( "Sys".COM.AlwaysOFF )
   END_RUNG
   RUNG wire#powerrail
      I_Contact( "Sys".COM.AlwaysON )
      S_Coil( "Sys".COM.AlwaysON )
   END_RUNG
   // the same network as SCL:
   IF "Sys".COM.AlwaysOFF THEN "Sys".COM.AlwaysOFF := FALSE; END_IF;
   IF NOT "Sys".COM.AlwaysON THEN "Sys".COM.AlwaysON := TRUE; END_IF;
END_REGION

REGION Network 2 (SCL): ScanTime
   // System Function don't modify
   "Sys".ScanTime.CyclePrevious := #OB1_PREV_CYCLE;
   "Sys".ScanTime.CycleMin := #OB1_MIN_CYCLE;
   "Sys".ScanTime.CycleMax := #OB1_MAX_CYCLE;
END_REGION

REGION Network 3: Hardware Clock Memory 0.1S
   // 系统程序段
   RUNG wire#powerrail
      Contact( "Sys".COM.AlwaysON )
      wire#w1
      Contact( "ClockMemory0.1s" )
      Coil( "Sys".COM.FlashTime100mS )
   END_RUNG
   RUNG wire#w1
      Contact( "ClockMemory0.2s" )
      Coil( "Sys".COM.FlashTime200mS )
   END_RUNG
   RUNG wire#w1
      Contact( "ClockMemory0.5s" )
      Coil( "Sys".COM.FlashTime500mS )
   END_RUNG
   RUNG wire#w1
      Contact( "ClockMemory1s" )
      Coil( "Sys".COM.FlashTime1S )
   END_RUNG
   RUNG wire#w1
      Contact( "ClockMemory2s" )
      Coil( "Sys".COM.FlashTime2S )
   END_RUNG
   // the same network as SCL:
   "Sys".COM.FlashTime100mS := "Sys".COM.AlwaysON AND "ClockMemory0.1s";
   "Sys".COM.FlashTime200mS := "Sys".COM.AlwaysON AND "ClockMemory0.2s";
   "Sys".COM.FlashTime500mS := "Sys".COM.AlwaysON AND "ClockMemory0.5s";
   "Sys".COM.FlashTime1S := "Sys".COM.AlwaysON AND "ClockMemory1s";
   "Sys".COM.FlashTime2S := "Sys".COM.AlwaysON AND "ClockMemory2s";
END_REGION

REGION Network 4: Date and time config
   // 系统程序段
   RUNG wire#powerrail
      Contact( "Sys".DateTime.Trigger )
      { S7_Templates := "date_type := Date_And_Time" } WR_SYS_T(IN := "Sys".DateTime.Set, RET_VAL => "Sys".RETVALI)
      R_Coil( "Sys".DateTime.Trigger )
   END_RUNG
   // the same network as SCL:
   "Sys".RETVALI := WR_SYS_T(EN := "Sys".DateTime.Trigger, IN := "Sys".DateTime.Set, ENO => #_w1);
   IF #_w1 THEN "Sys".DateTime.Trigger := FALSE; END_IF;
END_REGION

REGION Network 5: Diagnostic
   RUNG wire#powerrail
      "Diagnostic"(iCPUType := 2, iDBNum := 3001, iOffset := 132, iHardwareID := "Local~PROFINET_IO-System", oStatus => "DiagnosticDataBlock".Profinet.PNReadStatus)
   END_RUNG
   // the same network as SCL:
   "Diagnostic"(iCPUType := 2,
                iDBNum := 3001,
                iOffset := 132,
                iHardwareID := "Local~PROFINET_IO-System",
                oStatus => "DiagnosticDataBlock".Profinet.PNReadStatus);
END_REGION

REGION Network 6 (SCL): Win
       "ST10_GeneralData".HMI.Win.WinBullfer := 0;
       FOR #i := 1 TO 10 DO
           "ST10_GeneralData".HMI.Win.WinBullfer := "ST10_GeneralData".HMI.Win.WinBullfer + "ST10_GeneralData".HMI.Win."10x弹窗"[#i] * 11 +"ST10_GeneralData".HMI.Win."20x弹窗"[2] * 21 +"ST10_GeneralData".HMI.Win."30x弹窗"[#i] * 31 +"ST10_GeneralData".HMI.Win."40x弹窗"[#i] * 41;
       END_FOR;
       "ST10_GeneralData".HMI.Win.WinBullfer := ABS("ST10_GeneralData".HMI.Win.WinBullfer);
       "ST10_GeneralData".HMI.Win.TON[1](IN := "ST10_GeneralData".HMI.Win.Win <> "ST10_GeneralData".HMI.Win.WinBullfer,
                          PT := T#0.5S);
   IF "ST10_GeneralData".HMI.Win.TON[1].Q THEN
       "ST10_GeneralData".HMI.Win.Win := "ST10_GeneralData".HMI.Win.WinBullfer;
       END_IF;
END_REGION

REGION Network 7: MES_Shopworx
END_REGION

REGION Network 8: Call Main
   // 系统程序段
   RUNG wire#powerrail
      "ST10_Main"()
   END_RUNG
   // the same network as SCL:
   "ST10_Main"();
END_REGION

REGION Network 9: DataHandling in HMI
   RUNG wire#powerrail
      "AutoProcessDataPopUp_DB"(idx := "AutoProcess_HMI".IndexProcess)
   END_RUNG
   // the same network as SCL:
   "AutoProcessDataPopUp_DB"(idx := "AutoProcess_HMI".IndexProcess);   // "AutoProcessDataPopUp"
END_REGION

REGION Network 10: 上电初始化设备模式_手动模式 / Power-on Initialization Device Mode _ Manual mode
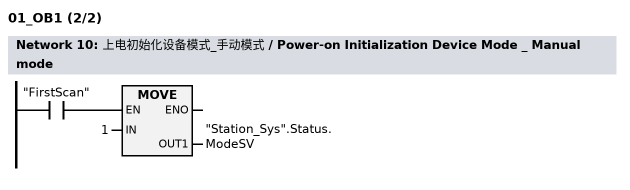
   RUNG wire#powerrail
      Contact( "FirstScan" )
      Move(in := 1, out1 => "Station_Sys".Status.ModeSV)
   END_RUNG
   // the same network as SCL:
   IF "FirstScan" THEN "Station_Sys".Status.ModeSV := 1; END_IF;
END_REGION
END_ORGANIZATION_BLOCK

FUNCTION "Diagnostic" : Void   // FC3001, SCL
TITLE = Diagnostic
{ S7_Optimized_Access := 'FALSE' }
AUTHOR : STD
FAMILY : RCS
VERSION : 18.0
// stored: AutoNumber false, SetENOAutomatically true
   VAR_INPUT
      iCPUType : Int;   // 1-DP&PN 2-PN
      iDBNum : Word;
      iOffset : Int;   // Start address
      iHardwareID : HW_IOSYSTEM;
   END_VAR
   VAR_OUTPUT
      oStatus : Int;
   END_VAR
   VAR_TEMP
      RDSRet : Struct
         Busy : Bool;
         Header : Struct
            Length : Word;
            Number : Word;
         END_STRUCT;
      END_STRUCT;
      retInt : Int;
      SSL : Struct
         SSID : Word;
         Index : Word;
         Length : Int;
      END_STRUCT;
      DR : Any;
      DRS AT DR : Struct
         SyntaxID : Byte;
         DataType : Byte;
         RepetitionFactor : Int;
         DB_Number : Word;
         MemoryAreaAddress : DWord;
      END_STRUCT;
   END_VAR
BEGIN

   (*############################################################
      RUHLAMAT SUZHOU ELEC.STD.
      Copyright (c) 2017. All rights reserved.    

      NAME OF FUNCTION BLOCK:         Diagnostic
      VERSION NUMBER:                 V3.0
      COMPOSER:                       Ming.Jiang

      CreateDate:                    16.Nov.2016
      ----------------------------------------------------------
      Interface description:
      IN:
          "iCPUType"
          iDBNum
          iOffset
          iHardwareID

      INOUT:
      OUT:
          oStatus

      ----------------------------------------------------------
      #RET_VALUE:

      #Alert Value:

      ----------------------------------------------------------
      Date           Name      Version           Activity                                                                              
      28.Nov.2016    JM        V3.0              add alarm

   ############################################################*)
   IF #iCPUType = 0 OR #iDBNum = 0 THEN
       ENO := 0;
       RETURN;
   ELSE
       IF #iCPUType=2 THEN
           GOTO PN;
       ELSIF #iCPUType=1 THEN
           ;
       ELSE
           ENO := 0;
           RETURN;
       END_IF;
       #DRS.SyntaxID := 16#10;
       #DRS.DataType := 16#02;
       #DRS.RepetitionFactor := 128;
       #DRS.DB_Number := #iDBNum;
       #DRS.MemoryAreaAddress := 16#8400_0000 OR (SHL(IN := INT_TO_DWORD(#iOffset), N := 3));
       #oStatus := DeviceStates(LADDR := #iHardwareID, MODE := 2, STATE := #DR);
   PN:
       #DRS.SyntaxID := 16#10;
       #DRS.DataType := 16#02;
       #DRS.RepetitionFactor := 128;
       #DRS.DB_Number := #iDBNum;
       #DRS.MemoryAreaAddress := 16#8400_0000 OR (SHL(IN := INT_TO_DWORD(#iOffset), N := 3));
       #oStatus := DeviceStates(LADDR := #iHardwareID, MODE := 2, STATE := #DR);
       // orginise interface data 
       ENO := 1;
       RETURN;
   END_IF;
END_FUNCTION

FUNCTION "ST10_Main" : Void   // FC1050, LAD
{ S7_Optimized_Access := 'FALSE' }
// stored: AutoNumber false, SetENOAutomatically false
BEGIN

REGION Network 1
   // 系统功能组调用部分
   // 1.该部分用户可以自己根据系统的组成将需要的功能块调用写在该部分
   // 2.该部分禁止与系统功能无关的程序在此处调用
END_REGION

NETWORK
TITLE = XXXX=====Station Relation/工位相关 =====StartXXXXX / XXXX=====Station Relation/Station correlation =====StartXXXXX

REGION Network 3: input /输入
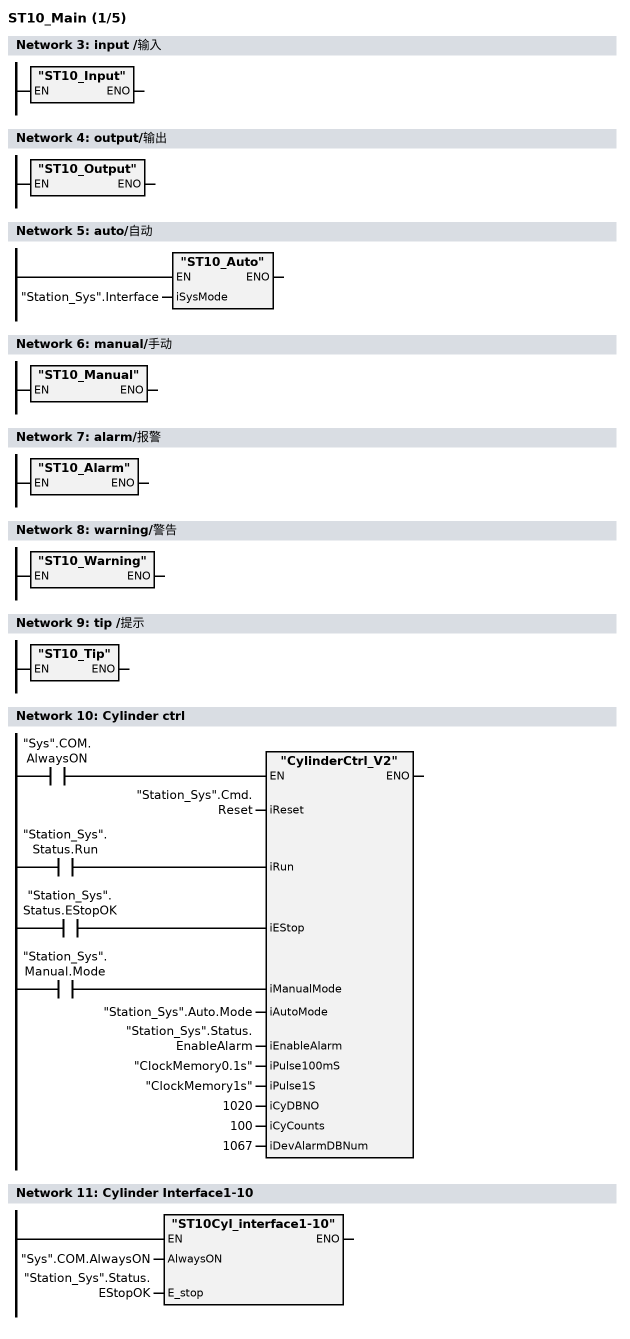
   RUNG wire#powerrail
      "ST10_Input"()
   END_RUNG
   // the same network as SCL:
   "ST10_Input"();
END_REGION

REGION Network 4: output/输出
   RUNG wire#powerrail
      "ST10_Output"()
   END_RUNG
   // the same network as SCL:
   "ST10_Output"();
END_REGION

REGION Network 5: auto/自动
   RUNG wire#powerrail
      "ST10_Auto"(iSysMode := "Station_Sys".Interface)
   END_RUNG
   // the same network as SCL:
   "ST10_Auto"(iSysMode := "Station_Sys".Interface);
END_REGION

REGION Network 6: manual/手动
   RUNG wire#powerrail
      "ST10_Manual"()
   END_RUNG
   // the same network as SCL:
   "ST10_Manual"();
END_REGION

REGION Network 7: alarm/报警
   RUNG wire#powerrail
      "ST10_Alarm"()
   END_RUNG
   // the same network as SCL:
   "ST10_Alarm"();
END_REGION

REGION Network 8: warning/警告
   RUNG wire#powerrail
      "ST10_Warning"()
   END_RUNG
   // the same network as SCL:
   "ST10_Warning"();
END_REGION

REGION Network 9: tip /提示
   RUNG wire#powerrail
      "ST10_Tip"()
   END_RUNG
   // the same network as SCL:
   "ST10_Tip"();
END_REGION

REGION Network 10: Cylinder ctrl
   RUNG wire#powerrail
      Contact( "Sys".COM.AlwaysON )
      "CylinderCtrl_V2"(iRun := wire#w1, iEStop := wire#w2, iManualMode := wire#w3, iReset := "Station_Sys".Cmd.Reset, iAutoMode := "Station_Sys".Auto.Mode, iEnableAlarm := "Station_Sys".Status.EnableAlarm, iPulse100mS := "ClockMemory0.1s", iPulse1S := "ClockMemory1s", iCyDBNO := 1020, iCyCounts := 100, iDevAlarmDBNum := 1067)
   END_RUNG
   RUNG wire#powerrail
      Contact( "Station_Sys".Status.Run )
   END_RUNG wire#w1
   RUNG wire#powerrail
      Contact( "Station_Sys".Status.EStopOK )
   END_RUNG wire#w2
   RUNG wire#powerrail
      Contact( "Station_Sys".Manual.Mode )
   END_RUNG wire#w3
   // the same network as SCL:
   IF "Sys".COM.AlwaysON THEN
       "CylinderCtrl_V2"(iReset := "Station_Sys".Cmd.Reset,
                         iRun := "Station_Sys".Status.Run,
                         iEStop := "Station_Sys".Status.EStopOK,
                         iManualMode := "Station_Sys".Manual.Mode,
                         iAutoMode := "Station_Sys".Auto.Mode,
                         iEnableAlarm := "Station_Sys".Status.EnableAlarm,
                         iPulse100mS := "ClockMemory0.1s",
                         iPulse1S := "ClockMemory1s",
                         iCyDBNO := 1020,
                         iCyCounts := 100,
                         iDevAlarmDBNum := 1067);
   END_IF;
END_REGION

REGION Network 11: Cylinder Interface1-10
   RUNG wire#powerrail
      "ST10Cyl_interface1-10"(AlwaysON := "Sys".COM.AlwaysON, E_stop := "Station_Sys".Status.EStopOK)
   END_RUNG
   // the same network as SCL:
   "ST10Cyl_interface1-10"(AlwaysON := "Sys".COM.AlwaysON, E_stop := "Station_Sys".Status.EStopOK);
END_REGION

REGION Network 12: Cylinder Interface11-20
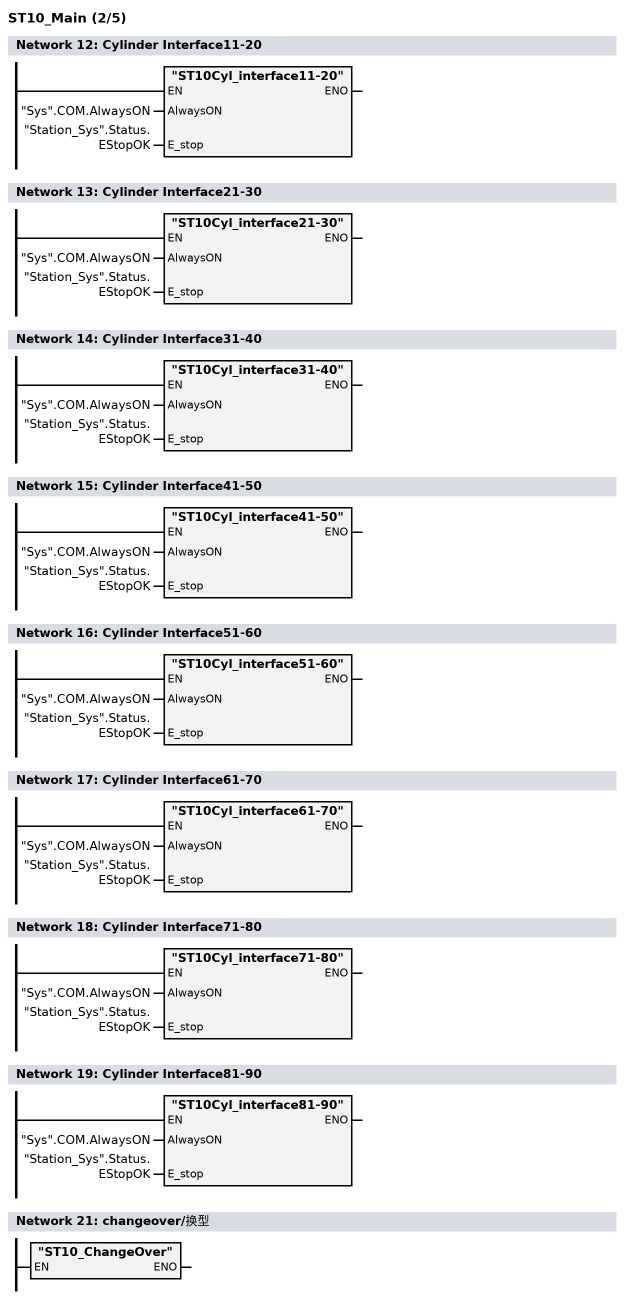
   RUNG wire#powerrail
      "ST10Cyl_interface11-20"(AlwaysON := "Sys".COM.AlwaysON, E_stop := "Station_Sys".Status.EStopOK)
   END_RUNG
   // the same network as SCL:
   "ST10Cyl_interface11-20"(AlwaysON := "Sys".COM.AlwaysON, E_stop := "Station_Sys".Status.EStopOK);
END_REGION

REGION Network 13: Cylinder Interface21-30
   RUNG wire#powerrail
      "ST10Cyl_interface21-30"(AlwaysON := "Sys".COM.AlwaysON, E_stop := "Station_Sys".Status.EStopOK)
   END_RUNG
   // the same network as SCL:
   "ST10Cyl_interface21-30"(AlwaysON := "Sys".COM.AlwaysON, E_stop := "Station_Sys".Status.EStopOK);
END_REGION

REGION Network 14: Cylinder Interface31-40
   RUNG wire#powerrail
      "ST10Cyl_interface31-40"(AlwaysON := "Sys".COM.AlwaysON, E_stop := "Station_Sys".Status.EStopOK)
   END_RUNG
   // the same network as SCL:
   "ST10Cyl_interface31-40"(AlwaysON := "Sys".COM.AlwaysON, E_stop := "Station_Sys".Status.EStopOK);
END_REGION

REGION Network 15: Cylinder Interface41-50
   RUNG wire#powerrail
      "ST10Cyl_interface41-50"(AlwaysON := "Sys".COM.AlwaysON, E_stop := "Station_Sys".Status.EStopOK)
   END_RUNG
   // the same network as SCL:
   "ST10Cyl_interface41-50"(AlwaysON := "Sys".COM.AlwaysON, E_stop := "Station_Sys".Status.EStopOK);
END_REGION

REGION Network 16: Cylinder Interface51-60
   RUNG wire#powerrail
      "ST10Cyl_interface51-60"(AlwaysON := "Sys".COM.AlwaysON, E_stop := "Station_Sys".Status.EStopOK)
   END_RUNG
   // the same network as SCL:
   "ST10Cyl_interface51-60"(AlwaysON := "Sys".COM.AlwaysON, E_stop := "Station_Sys".Status.EStopOK);
END_REGION

REGION Network 17: Cylinder Interface61-70
   RUNG wire#powerrail
      "ST10Cyl_interface61-70"(AlwaysON := "Sys".COM.AlwaysON, E_stop := "Station_Sys".Status.EStopOK)
   END_RUNG
   // the same network as SCL:
   "ST10Cyl_interface61-70"(AlwaysON := "Sys".COM.AlwaysON, E_stop := "Station_Sys".Status.EStopOK);
END_REGION

REGION Network 18: Cylinder Interface71-80
   RUNG wire#powerrail
      "ST10Cyl_interface71-80"(AlwaysON := "Sys".COM.AlwaysON, E_stop := "Station_Sys".Status.EStopOK)
   END_RUNG
   // the same network as SCL:
   "ST10Cyl_interface71-80"(AlwaysON := "Sys".COM.AlwaysON, E_stop := "Station_Sys".Status.EStopOK);
END_REGION

REGION Network 19: Cylinder Interface81-90
   RUNG wire#powerrail
      "ST10Cyl_interface81-90"(AlwaysON := "Sys".COM.AlwaysON, E_stop := "Station_Sys".Status.EStopOK)
   END_RUNG
   // the same network as SCL:
   "ST10Cyl_interface81-90"(AlwaysON := "Sys".COM.AlwaysON, E_stop := "Station_Sys".Status.EStopOK);
END_REGION

REGION Network 21: changeover/换型
   RUNG wire#powerrail
      "ST10_ChangeOver"()
   END_RUNG
   // the same network as SCL:
   "ST10_ChangeOver"();
END_REGION

REGION Network 22: Device
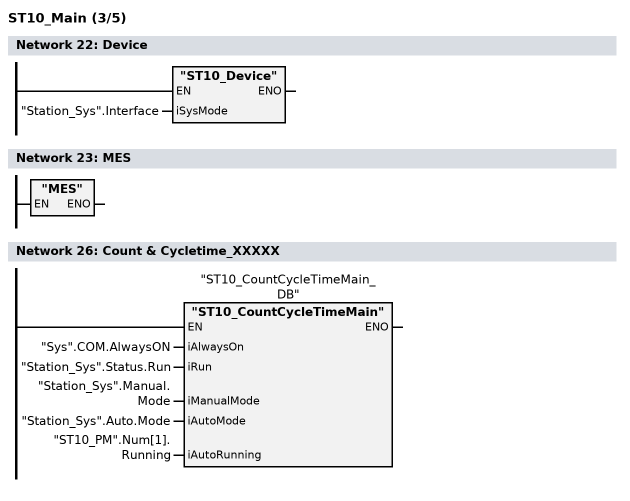
   RUNG wire#powerrail
      "ST10_Device"(iSysMode := "Station_Sys".Interface)
   END_RUNG
   // the same network as SCL:
   "ST10_Device"(iSysMode := "Station_Sys".Interface);
END_REGION

REGION Network 23: MES
   RUNG wire#powerrail
      "MES"()
   END_RUNG
   // the same network as SCL:
   "MES"();
END_REGION

REGION Network 24: =====System Function related information Section =====Start
END_REGION

NETWORK
TITLE = SystemFunction IO

REGION Network 26: Count & Cycletime_XXXXX
   RUNG wire#powerrail
      "ST10_CountCycleTimeMain_DB"(iAlwaysOn := "Sys".COM.AlwaysON, iRun := "Station_Sys".Status.Run, iManualMode := "Station_Sys".Manual.Mode, iAutoMode := "Station_Sys".Auto.Mode, iAutoRunning := "ST10_PM".Num[1].Running)
   END_RUNG
   // the same network as SCL:
   "ST10_CountCycleTimeMain_DB"(iAlwaysOn := "Sys".COM.AlwaysON,   // "ST10_CountCycleTimeMain"
                           iRun := "Station_Sys".Status.Run,
                           iManualMode := "Station_Sys".Manual.Mode,
                           iAutoMode := "Station_Sys".Auto.Mode,
                           iAutoRunning := "ST10_PM".Num[1].Running);
END_REGION

REGION Network 27: System mode
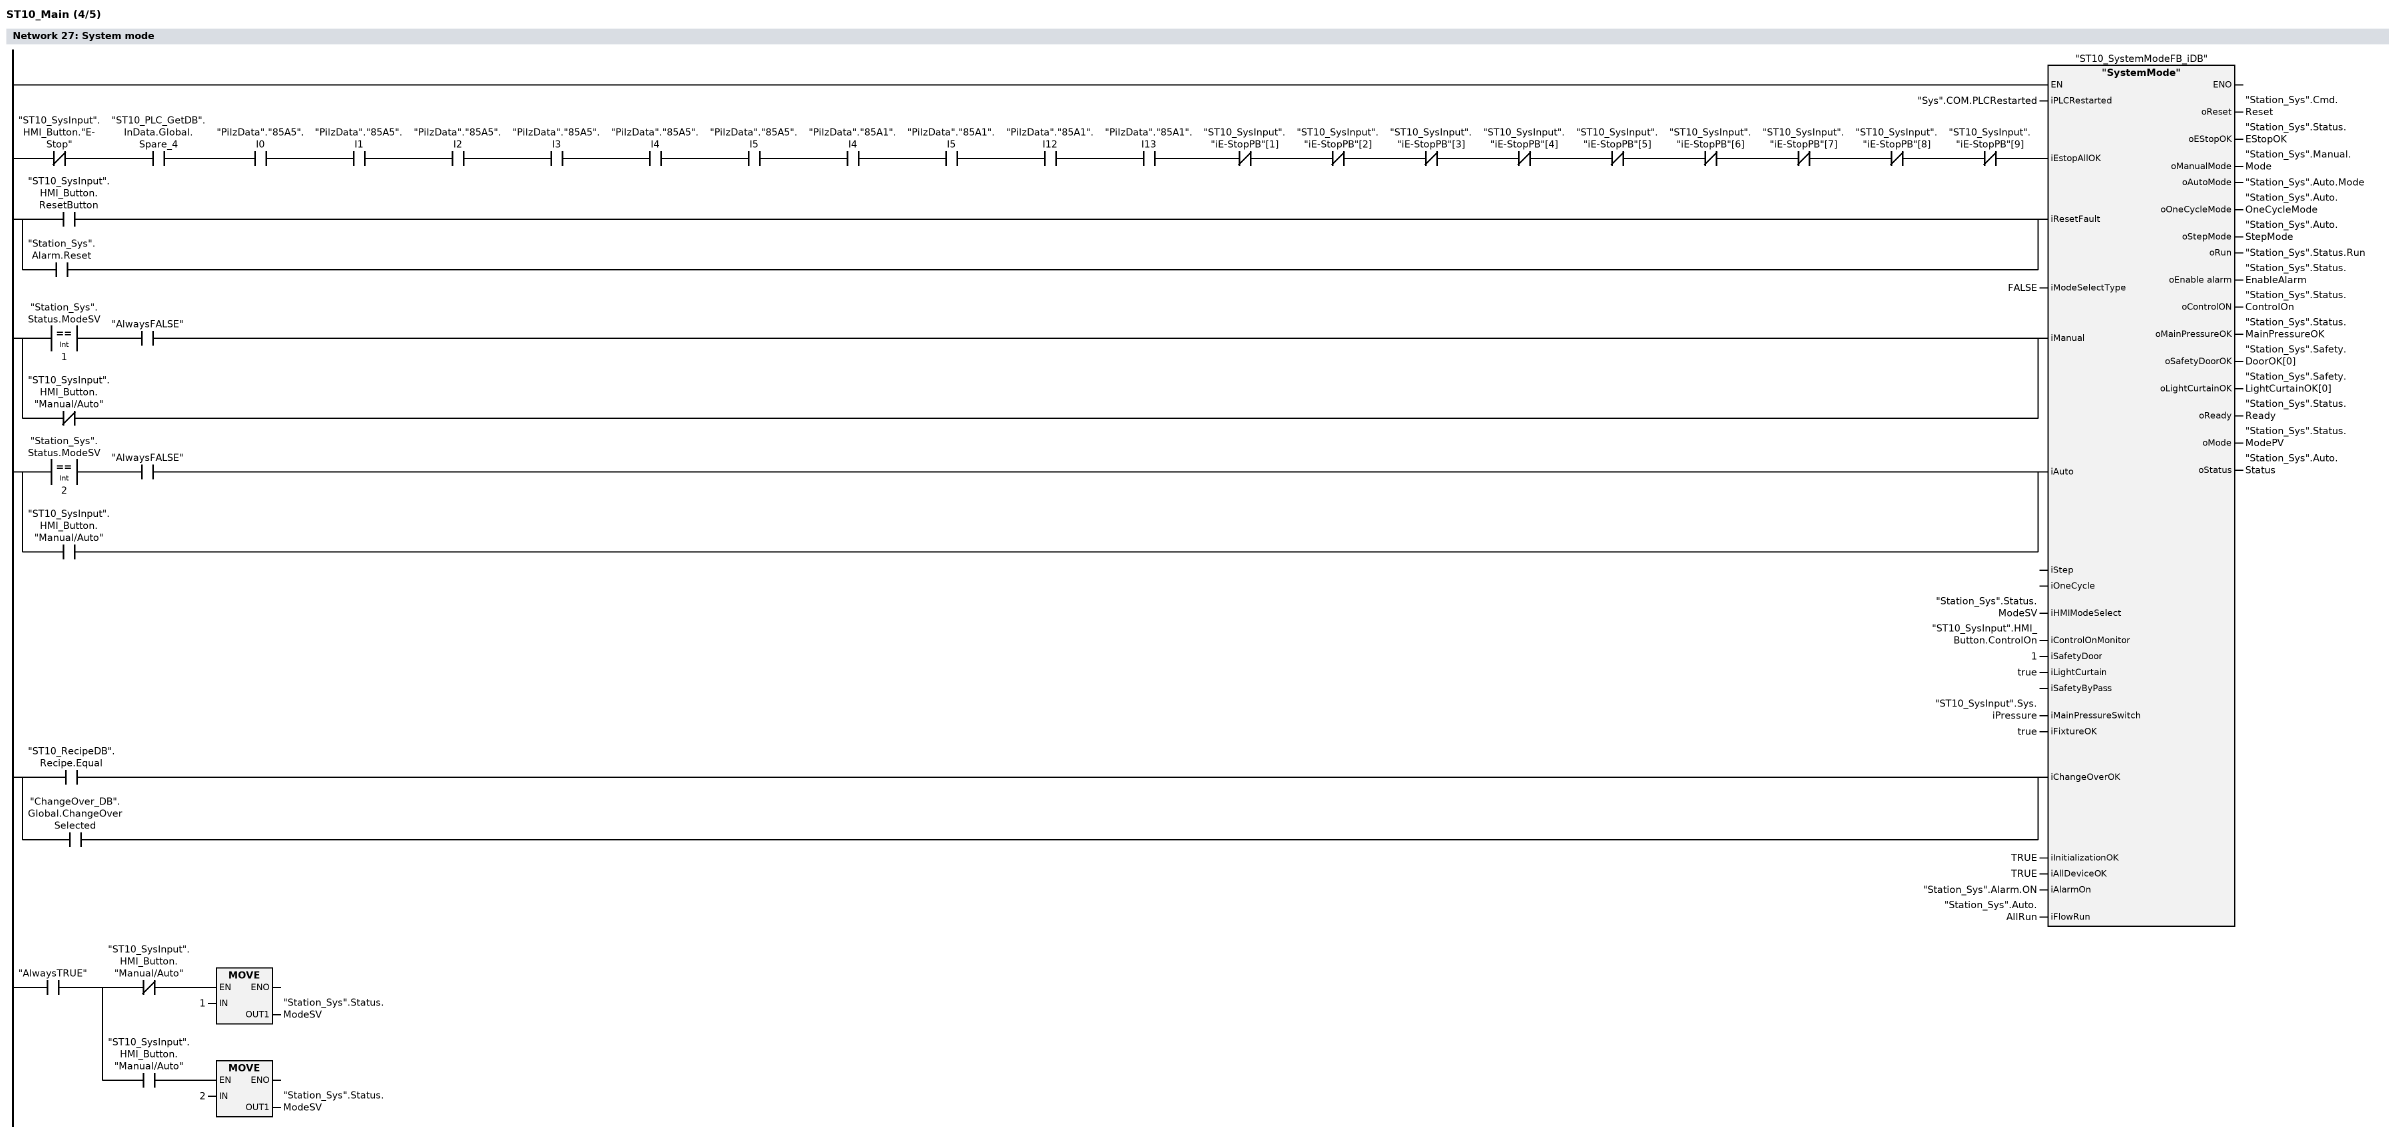
   RUNG wire#powerrail
      "ST10_SystemModeFB_iDB"(iEstopAllOK := wire#w1, iResetFault := wire#w2, iManual := wire#w3, iAuto := wire#w4, iChangeOverOK := wire#w5, iPLCRestarted := "Sys".COM.PLCRestarted, iModeSelectType := FALSE, iStep :=, iOneCycle :=, iHMIModeSelect := "Station_Sys".Status.ModeSV, iControlOnMonitor := "ST10_SysInput".HMI_Button.ControlOn, iSafetyDoor := 1, iLightCurtain := true, iSafetyByPass :=, iMainPressureSwitch := "ST10_SysInput".Sys.iPressure, iFixtureOK := true, iInitializationOK := TRUE, iAllDeviceOK := TRUE, iAlarmOn := "Station_Sys".Alarm.ON, iFlowRun := "Station_Sys".Auto.AllRun, oReset => "Station_Sys".Cmd.Reset, oEStopOK => "Station_Sys".Status.EStopOK, oManualMode => "Station_Sys".Manual.Mode, oAutoMode => "Station_Sys".Auto.Mode, oOneCycleMode => "Station_Sys".Auto.OneCycleMode, oStepMode => "Station_Sys".Auto.StepMode, oRun => "Station_Sys".Status.Run, "oEnable alarm" => "Station_Sys".Status.EnableAlarm, oControlON => "Station_Sys".Status.ControlOn, oMainPressureOK => "Station_Sys".Status.MainPressureOK, oSafetyDoorOK => "Station_Sys".Safety.DoorOK[0], oLightCurtainOK => "Station_Sys".Safety.LightCurtainOK[0], oReady => "Station_Sys".Status.Ready, oMode => "Station_Sys".Status.ModePV, oStatus => "Station_Sys".Auto.Status)
   END_RUNG
   RUNG wire#powerrail
      I_Contact( "ST10_SysInput".HMI_Button."E-Stop" )
      Contact( "ST10_PLC_GetDB".InData.Global.Spare_4 )
      Contact( "PilzData"."85A5".I0 )
      Contact( "PilzData"."85A5".I1 )
      Contact( "PilzData"."85A5".I2 )
      Contact( "PilzData"."85A5".I3 )
      Contact( "PilzData"."85A5".I4 )
      Contact( "PilzData"."85A5".I5 )
      Contact( "PilzData"."85A1".I4 )
      Contact( "PilzData"."85A1".I5 )
      Contact( "PilzData"."85A1".I12 )
      Contact( "PilzData"."85A1".I13 )
      I_Contact( "ST10_SysInput"."iE-StopPB"[1] )
      I_Contact( "ST10_SysInput"."iE-StopPB"[2] )
      I_Contact( "ST10_SysInput"."iE-StopPB"[3] )
      I_Contact( "ST10_SysInput"."iE-StopPB"[4] )
      I_Contact( "ST10_SysInput"."iE-StopPB"[5] )
      I_Contact( "ST10_SysInput"."iE-StopPB"[6] )
      I_Contact( "ST10_SysInput"."iE-StopPB"[7] )
      I_Contact( "ST10_SysInput"."iE-StopPB"[8] )
      I_Contact( "ST10_SysInput"."iE-StopPB"[9] )
   END_RUNG wire#w1
   RUNG wire#powerrail
      Contact( "ST10_SysInput".HMI_Button.ResetButton )
   END_RUNG wire#w2
   RUNG wire#powerrail
      Contact( "Station_Sys".Alarm.Reset )
   END_RUNG wire#w2
   RUNG wire#powerrail
      { S7_Templates := "SrcType := Int" } EQ_Contact(in1 := "Station_Sys".Status.ModeSV, in2 := 1)
      Contact( "AlwaysFALSE" )
   END_RUNG wire#w3
   RUNG wire#powerrail
      I_Contact( "ST10_SysInput".HMI_Button."Manual/Auto" )
   END_RUNG wire#w3
   RUNG wire#powerrail
      { S7_Templates := "SrcType := Int" } EQ_Contact(in1 := "Station_Sys".Status.ModeSV, in2 := 2)
      Contact( "AlwaysFALSE" )
   END_RUNG wire#w4
   RUNG wire#powerrail
      Contact( "ST10_SysInput".HMI_Button."Manual/Auto" )
   END_RUNG wire#w4
   RUNG wire#powerrail
      Contact( "ST10_RecipeDB".Recipe.Equal )
   END_RUNG wire#w5
   RUNG wire#powerrail
      Contact( "ChangeOver_DB".Global.ChangeOverSelected )
   END_RUNG wire#w5
   RUNG wire#powerrail
      Contact( "AlwaysTRUE" )
      wire#w6
      I_Contact( "ST10_SysInput".HMI_Button."Manual/Auto" )
      Move(in := 1, out1 => "Station_Sys".Status.ModeSV)
   END_RUNG
   RUNG wire#w6
      Contact( "ST10_SysInput".HMI_Button."Manual/Auto" )
      Move(in := 2, out1 => "Station_Sys".Status.ModeSV)
   END_RUNG
   // the same network as SCL:
   "ST10_SystemModeFB_iDB"(iPLCRestarted := "Sys".COM.PLCRestarted,   // "SystemMode"
                           iEstopAllOK := NOT "ST10_SysInput".HMI_Button."E-Stop" AND "ST10_PLC_GetDB".InData.Global.Spare_4 AND "PilzData"."85A5".I0 AND "PilzData"."85A5".I1 AND "PilzData"."85A5".I2 AND "PilzData"."85A5".I3 AND "PilzData"."85A5".I4 AND "PilzData"."85A5".I5 AND "PilzData"."85A1".I4 AND "PilzData"."85A1".I5 AND "PilzData"."85A1".I12 AND "PilzData"."85A1".I13 AND NOT "ST10_SysInput"."iE-StopPB"[1] AND NOT "ST10_SysInput"."iE-StopPB"[2] AND NOT "ST10_SysInput"."iE-StopPB"[3] AND NOT "ST10_SysInput"."iE-StopPB"[4] AND NOT "ST10_SysInput"."iE-StopPB"[5] AND NOT "ST10_SysInput"."iE-StopPB"[6] AND NOT "ST10_SysInput"."iE-StopPB"[7] AND NOT "ST10_SysInput"."iE-StopPB"[8] AND NOT "ST10_SysInput"."iE-StopPB"[9],
                           iResetFault := "ST10_SysInput".HMI_Button.ResetButton OR "Station_Sys".Alarm.Reset,
                           iModeSelectType := FALSE,
                           iManual := (("Station_Sys".Status.ModeSV = 1) AND "AlwaysFALSE") OR NOT "ST10_SysInput".HMI_Button."Manual/Auto",
                           iAuto := (("Station_Sys".Status.ModeSV = 2) AND "AlwaysFALSE") OR "ST10_SysInput".HMI_Button."Manual/Auto",
                           iHMIModeSelect := "Station_Sys".Status.ModeSV,
                           iControlOnMonitor := "ST10_SysInput".HMI_Button.ControlOn,
                           iSafetyDoor := 1,
                           iLightCurtain := true,
                           iMainPressureSwitch := "ST10_SysInput".Sys.iPressure,
                           iFixtureOK := true,
                           iChangeOverOK := "ST10_RecipeDB".Recipe.Equal OR "ChangeOver_DB".Global.ChangeOverSelected,
                           iInitializationOK := TRUE,
                           iAllDeviceOK := TRUE,
                           iAlarmOn := "Station_Sys".Alarm.ON,
                           iFlowRun := "Station_Sys".Auto.AllRun,
                           oReset => "Station_Sys".Cmd.Reset,
                           oEStopOK => "Station_Sys".Status.EStopOK,
                           oManualMode => "Station_Sys".Manual.Mode,
                           oAutoMode => "Station_Sys".Auto.Mode,
                           oOneCycleMode => "Station_Sys".Auto.OneCycleMode,
                           oStepMode => "Station_Sys".Auto.StepMode,
                           oRun => "Station_Sys".Status.Run,
                           "oEnable alarm" => "Station_Sys".Status.EnableAlarm,
                           oControlON => "Station_Sys".Status.ControlOn,
                           oMainPressureOK => "Station_Sys".Status.MainPressureOK,
                           oSafetyDoorOK => "Station_Sys".Safety.DoorOK[0],
                           oLightCurtainOK => "Station_Sys".Safety.LightCurtainOK[0],
                           oReady => "Station_Sys".Status.Ready,
                           oMode => "Station_Sys".Status.ModePV,
                           oStatus => "Station_Sys".Auto.Status);
   IF "AlwaysTRUE" AND NOT "ST10_SysInput".HMI_Button."Manual/Auto" THEN
       "Station_Sys".Status.ModeSV := 1;
   END_IF;
   IF "AlwaysTRUE" AND "ST10_SysInput".HMI_Button."Manual/Auto" THEN
       "Station_Sys".Status.ModeSV := 2;
   END_IF;
END_REGION

REGION Network 28: Start button
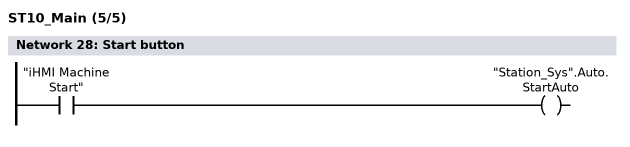
   RUNG wire#powerrail
      Contact( "iHMI Machine Start" )
      Coil( "Station_Sys".Auto.StartAuto )
   END_RUNG
   // the same network as SCL:
   "Station_Sys".Auto.StartAuto := "iHMI Machine Start";
END_REGION

REGION Network 29 (SCL): System Interface
   "Station_Sys".Interface.CPUFristCycle  := "Sys".COM.PLCRestarted;
   "Station_Sys".Interface.SysRun         := "Station_Sys".Status.Run;
   "Station_Sys".Interface.Reset          := "Station_Sys".Cmd.Reset;
   "Station_Sys".Interface.EstopOK        := "Station_Sys".Status.EStopOK;
   "Station_Sys".Interface.SafetyDoorOK   := "Station_Sys".Safety.DoorOK[0];
   "Station_Sys".Interface.LightCurtainOK := "Station_Sys".Safety.LightCurtainOK[0];
   "Station_Sys".Interface.SetInitial     := "Station_Sys".Initial.Set;
   "Station_Sys".Interface.InitialRun     := "Station_Sys".Initial.Running;
   "Station_Sys".Interface.Ready          := "Station_Sys".Status.Ready;
   "Station_Sys".Interface.ManualMode     := "Station_Sys".Manual.Mode;
   "Station_Sys".Interface.Auto           := "Station_Sys".Auto;
END_REGION

REGION Network 30: =====System Function related information Section =====End
END_REGION

REGION Network 31: CallCalibration//标定调用
END_REGION

REGION Network 32 (SCL): ByPass Button
   // A
   "ST10_GeneralData".FunctionDeSelect.A.FunctionDeSelected_Servo380A1  := "ST10_GeneralData".FunctionDeSelect.A.DeSelectPB_Servo380A1;
   "ST10_GeneralData".FunctionDeSelect.A.FunctionDeSelected_Servo381A1  := "ST10_GeneralData".FunctionDeSelect.A.DeSelectPB_Servo381A1;
   "ST10_GeneralData".FunctionDeSelect.A.FunctionDeSelected_Servo383A1  := "ST10_GeneralData".FunctionDeSelect.A.DeSelectPB_Servo383A1;
   "ST10_GeneralData".FunctionDeSelect.A.FunctionDeSelected_Reader800A1 := "ST10_GeneralData".FunctionDeSelect.A.DeSelectPB_Reader800A1;
   "ST10_GeneralData".FunctionDeSelect.A.FunctionDeSelected_Reader801A1 := "ST10_GeneralData".FunctionDeSelect.A.DeSelectPB_Reader801A1;
   "ST10_GeneralData".FunctionDeSelect.A.FunctionDeSelected_Reader802A1 := "ST10_GeneralData".FunctionDeSelect.A.DeSelectPB_Reader802A1;
   "ST10_GeneralData".FunctionDeSelect.A.FunctionDeSelected_Reader803A1 := "ST10_GeneralData".FunctionDeSelect.A.DeSelectPB_Reader803A1;
   "ST10_GeneralData".FunctionDeSelect.A.FunctionDeSelected_Reader804A1 := "ST10_GeneralData".FunctionDeSelect.A.DeSelectPB_Reader804A1;

   // B
   "ST10_GeneralData".FunctionDeSelect.B.FunctionDeSelected_Press372A1     := "ST10_GeneralData".FunctionDeSelect.B.DeSelectPB_Press372A1;
   "ST10_GeneralData".FunctionDeSelect.B.FunctionDeSelected_Press375A1     := "ST10_GeneralData".FunctionDeSelect.B.DeSelectPB_Press375A1;
   "ST10_GeneralData".FunctionDeSelect.B.FunctionDeSelected_Reader806A1    := "ST10_GeneralData".FunctionDeSelect.B.DeSelectPB_Reader806A1;
   "ST10_GeneralData".FunctionDeSelect.B.FunctionDeSelected_TestPress372A1 := "ST10_GeneralData".FunctionDeSelect.B.DeSelectPB_TestPress372A1;
   "ST10_GeneralData".FunctionDeSelect.B.FunctionDeSelected_TestPress375A1 := "ST10_GeneralData".FunctionDeSelect.B.DeSelectPB_TestPress375A1;

   // C
   "ST10_GeneralData".FunctionDeSelect.C.FunctionDeSelected_Servo382A1 := "ST10_GeneralData".FunctionDeSelect.C.DeSelectPB_Servo382A1;
   "ST10_GeneralData".FunctionDeSelect.C.FunctionDeSelected_ServoIAI := "ST10_GeneralData".FunctionDeSelect.C.DeSelectPB_ServoIAI;
   "ST10_GeneralData".FunctionDeSelect.C.FunctionDeSelected_IV3810A1 := "ST10_GeneralData".FunctionDeSelect.C.DeSelectPB_IV3810A1;
   "ST10_GeneralData".FunctionDeSelect.C.FunctionDeSelected_IV3811A1 := "ST10_GeneralData".FunctionDeSelect.C.DeSelectPB_IV3811A1;
   "ST10_GeneralData".FunctionDeSelect.C.FunctionDeSelected_Glue := "ST10_GeneralData".FunctionDeSelect.C.DeSelectPB_Glue;

   // E
   "ST10_GeneralData".FunctionDeSelect.E.FunctionDeSelected := "ST10_GeneralData".FunctionDeSelect.E.DeSelectPB;

   // F
   "ST10_GeneralData".FunctionDeSelect.F.FunctionDeSelected_Reader805A1 := "ST10_GeneralData".FunctionDeSelect.F.DeSelectPB_Reader805A1;

   // H
   "ST10_GeneralData".FunctionDeSelect.H.FunctionDeSelected := "ST10_GeneralData".FunctionDeSelect.H.DeSelectPB;

   // J
   "ST10_GeneralData".FunctionDeSelect.J.FunctionDeSelected := "ST10_GeneralData".FunctionDeSelect.J.DeSelectPB;

   // K
   "ST10_GeneralData".FunctionDeSelect.K.FunctionDeSelected := "ST10_GeneralData".FunctionDeSelect.K.DeSelectPB;

   // L
   "ST10_GeneralData".FunctionDeSelect.L.FunctionDeSelected := "ST10_GeneralData".FunctionDeSelect.L.DeSelectPB;

   // MES
   "ST10_GeneralData".FunctionDeSelect.MES.FunctionDeSelected := "ST10_GeneralData".FunctionDeSelect.MES.DeSelectPB;

   //Auto>Maanual  ScanFixture
   "ST10_GeneralData".FunctionDeSelect.Global.FunctionDeSelected_ScanFixture := "ST10_GeneralData".FunctionDeSelect.Global.DeSelectPB_ScanFixture;
END_REGION
END_FUNCTION

FUNCTION "ST10_Input" : Void   // FC1001, LAD
{ S7_Optimized_Access := 'FALSE' }
// 注：本程序用来处理需要滤波，延时、计算的输入信号
// stored: AutoNumber false, SetENOAutomatically false
BEGIN

REGION Network 1 (SCL): HMI信号映射 / HMI signal mapping
   "ST10_SysInput".HMI_Button.ControlOn := "iHMI Control On";
   //"ST350_SysInput".HMI_Button.ControlOff:=
   "ST10_SysInput".HMI_Button.MachineStart := "iHMI Machine Start";
   "ST10_SysInput".HMI_Button.MachineStop := "iHMI Machine Stop";
   "ST10_SysInput".HMI_Button.ResetButton := "iHMI ResetButton";
   "ST10_SysInput".HMI_Button."Manual/Auto" := "iHMI Manual/Auto";
   "ST10_SysInput".HMI_Button.SafetyGateUnlock := "iHMI Safety Gate Unlock";
   "ST10_SysInput".HMI_Button."E-Stop" :=  "iHMI E-Stop";
END_REGION

REGION Network 2 (SCL): Sys IO Image
   "ST10_SysInput".Sys.iCircuitBreakerOK1 := "iCircuit Breaker OK_1";
   "ST10_SysInput".Sys.iCircuitBreakerOK2 := "iCircuit Breaker OK_2";
   "ST10_SysInput".Sys.iPressure:= "iPressure";
END_REGION

REGION Network 3 (SCL): iE-StopPB
   "ST10_SysInput"."iE-StopPB"[1] := "iE_StopButton2_A01";
   "ST10_SysInput"."iE-StopPB"[2] := "iE_StopButton3_A02";
   "ST10_SysInput"."iE-StopPB"[3] := "iE_StopButton4_H";
   "ST10_SysInput"."iE-StopPB"[4] := "iE_StopButton5_J";
   "ST10_SysInput"."iE-StopPB"[5] := "iE_StopButton6_K";
   "ST10_SysInput"."iE-StopPB"[6] := "iE_StopButton7_L";
   "ST10_SysInput"."iE-StopPB"[7] := "iH_StopButton";
   "ST10_SysInput"."iE-StopPB"[8] := "iJ_StopButton";
   "ST10_SysInput"."iE-StopPB"[9] := "iK_StopButton";
END_REGION

REGION Network 4 (SCL): iSafetyGatFeedBack
   (*
   "ST350_SysInput".iSafetyGatFeedBack[1] := "iSafety door Locking FeedBack_1";
   "ST350_SysInput".iSafetyGatFeedBack[2] := "iSafety door Locking FeedBack_2";
   "ST350_SysInput".iSafetyGatFeedBack[3] := "iSafety door Locking FeedBack_3";
   "ST350_SysInput".iSafetyGatFeedBack[4] := "iSafety door Locking FeedBack_4";
   "ST350_SysInput".iSafetyGatFeedBack[5] := "iSafety door Locking FeedBack_5";
   "ST350_SysInput".iSafetyGatFeedBack[6] := "iSafety door Locking FeedBack_6";
   "ST350_SysInput".iSafetyGatFeedBack[7] := "iSafety door Locking FeedBack_7";
   "ST350_SysInput".iSafetyGatFeedBack[8] := "iSafety door Locking FeedBack_8";
   *)
END_REGION

REGION Network 5 (SCL): iSafetydoorLockingFeedBack
   "ST10_SysInput".iSafetydoorLockingFeedBack[1] := "iSafety door Locking FeedBack_1";
   "ST10_SysInput".iSafetydoorLockingFeedBack[2] := "iSafety door Locking FeedBack_2";
   "ST10_SysInput".iSafetydoorLockingFeedBack[3] := "iSafety door Locking FeedBack_3";
   "ST10_SysInput".iSafetydoorLockingFeedBack[4] := "iSafety door Locking FeedBack_4";
   "ST10_SysInput".iSafetydoorLockingFeedBack[5] := "iSafety door Locking FeedBack_5";
   "ST10_SysInput".iSafetydoorLockingFeedBack[6] := "iSafety door Locking FeedBack_6";
   "ST10_SysInput".iSafetydoorLockingFeedBack[7] := "iSafety door Locking FeedBack_7";
   "ST10_SysInput".iSafetydoorLockingFeedBack[8] := "iSafety door Locking FeedBack_8";
END_REGION

REGION Network 6 (SCL): iSafetydoorLockingFeedBack
   "ST10_SysInput".iMaterieldoorLockingFeedBack[1] := "iMateriel Door Locking FeedBack_H1";
   "ST10_SysInput".iMaterieldoorLockingFeedBack[2] := "iMateriel Door Locking FeedBack_H2";
   "ST10_SysInput".iMaterieldoorLockingFeedBack[3] := "iMateriel Door Locking FeedBack_J1";
   "ST10_SysInput".iMaterieldoorLockingFeedBack[4] := "iMateriel Door Locking FeedBack_J2";
   "ST10_SysInput".iMaterieldoorLockingFeedBack[5] := "iMateriel Door Locking FeedBack_K1";
   "ST10_SysInput".iMaterieldoorLockingFeedBack[6] := "iMateriel Door Locking FeedBack_K2";
   "ST10_SysInput".iMaterieldoorLockingFeedBack[7] := "iMateriel Door Locking FeedBack_L1";
END_REGION
END_FUNCTION

FUNCTION "ST10_Output" : Void   // FC1002, LAD
{ S7_Optimized_Access := 'FALSE' }
// stored: AutoNumber false, SetENOAutomatically false
   VAR_TEMP   // added for the SCL form of the ladder/FBD networks
      _w1 : Bool;
      _w2 : Bool;
      _w3 : Bool;
      _w4 : Bool;
      _w5 : Bool;
      _w6 : Bool;
   END_VAR
BEGIN

REGION Network 1 (SCL): 安全门锁定信号映射SafetyDoorCoil / Safety door lock signal mapping //SafetyDoorCoil
   "oSafetyDoorLocked_1" := "ST10_SysOutput".SafetyDoorCoil[1];
   "oSafetyDoorLocked_2" := "ST10_SysOutput".SafetyDoorCoil[2];
   "oSafetyDoorLocked_3" := "ST10_SysOutput".SafetyDoorCoil[3];
   "oSafetyDoorLocked_4" := "ST10_SysOutput".SafetyDoorCoil[4];
   "oSafetyDoorLocked_5" := "ST10_SysOutput".SafetyDoorCoil[5];
   "oSafetyDoorLocked_6" := "ST10_SysOutput".SafetyDoorCoil[6];
   "oSafetyDoorLocked_7" := "ST10_SysOutput".SafetyDoorCoil[7];
   "oSafetyDoorLocked_8" := "ST10_SysOutput".SafetyDoorCoil[8];
   "oSafetyDoorLocked" := "ST10_SysOutput".SafetyDoorCoil[9];
END_REGION

REGION Network 2 (SCL): 安全门锁定信号映射SafetyDoorCoil / Safety door lock signal mapping //SafetyDoorCoil
   "oMaterielDoorLocked_H1" := "ST10_SysOutput".MaterialDoorCoil[1];
   "oMaterielDoorLocked_H2" := "ST10_SysOutput".MaterialDoorCoil[2];
   "oMaterielDoorLocked_J1" := "ST10_SysOutput".MaterialDoorCoil[3];
   "oMaterielDoorLocked_J2" := "ST10_SysOutput".MaterialDoorCoil[4];
   "oMaterielDoorLocked_K1" := "ST10_SysOutput".MaterialDoorCoil[5];
   "oMaterielDoorLocked_K2" := "ST10_SysOutput".MaterialDoorCoil[6];
   "oMaterielDoorLocked_L1" := "ST10_SysOutput".MaterialDoorCoil[7];


   "oE-NG-01SafetyGate" := "ST10_SysOutput".MaterialDoorCoil[8];
   "oE-NG-02SafetyGate" := "ST10_SysOutput".MaterialDoorCoil[9];
END_REGION

REGION Network 3: 塔灯 / Tower light
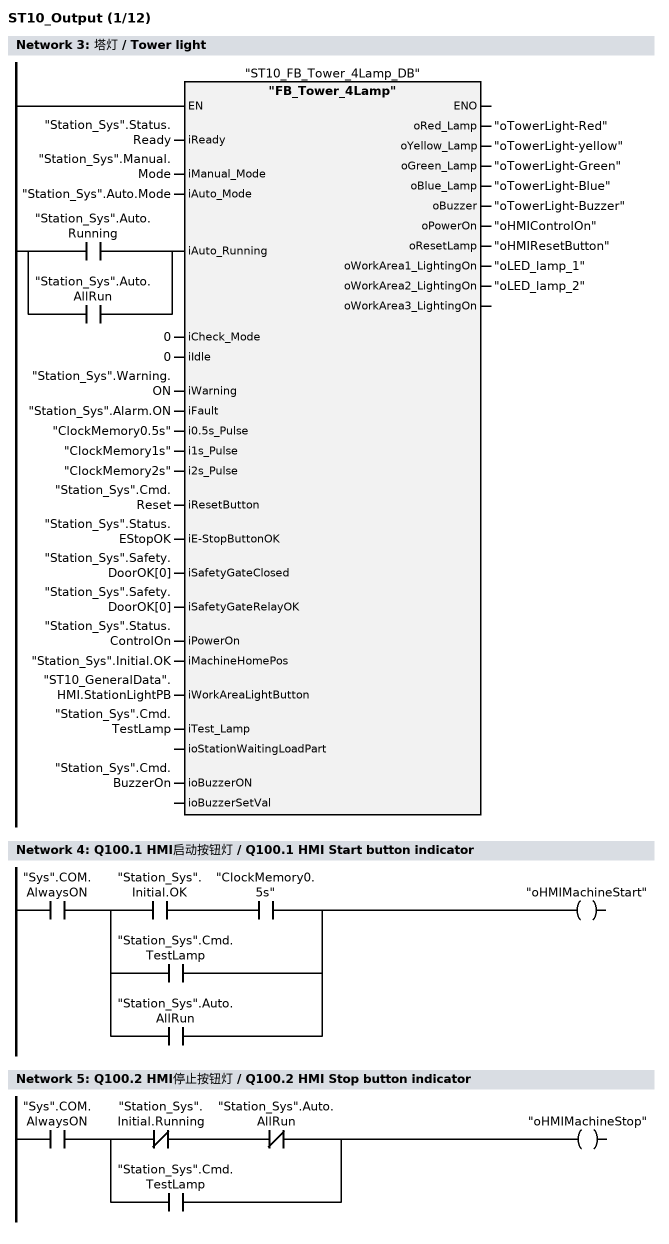
   RUNG wire#powerrail
      "ST10_FB_Tower_4Lamp_DB"(iAuto_Running := wire#w1, iReady := "Station_Sys".Status.Ready, iManual_Mode := "Station_Sys".Manual.Mode, iAuto_Mode := "Station_Sys".Auto.Mode, iCheck_Mode := 0, iIdle := 0, iWarning := "Station_Sys".Warning.ON, iFault := "Station_Sys".Alarm.ON, "i0.5s_Pulse" := "ClockMemory0.5s", i1s_Pulse := "ClockMemory1s", i2s_Pulse := "ClockMemory2s", iResetButton := "Station_Sys".Cmd.Reset, "iE-StopButtonOK" := "Station_Sys".Status.EStopOK, iSafetyGateClosed := "Station_Sys".Safety.DoorOK[0], iSafetyGateRelayOK := "Station_Sys".Safety.DoorOK[0], iPowerOn := "Station_Sys".Status.ControlOn, iMachineHomePos := "Station_Sys".Initial.OK, iWorkAreaLightButton := "ST10_GeneralData".HMI.StationLightPB, iTest_Lamp := "Station_Sys".Cmd.TestLamp, ioStationWaitingLoadPart :=, ioBuzzerON := "Station_Sys".Cmd.BuzzerOn, ioBuzzerSetVal :=, oRed_Lamp => "oTowerLight-Red", oYellow_Lamp => "oTowerLight-yellow", oGreen_Lamp => "oTowerLight-Green", oBlue_Lamp => "oTowerLight-Blue", oBuzzer => "oTowerLight-Buzzer", oPowerOn => "oHMIControlOn", oResetLamp => "oHMIResetButton", oWorkArea1_LightingOn => "oLED_lamp_1", oWorkArea2_LightingOn => "oLED_lamp_2", oWorkArea3_LightingOn =>)
   END_RUNG
   RUNG wire#powerrail
      Contact( "Station_Sys".Auto.Running )
   END_RUNG wire#w1
   RUNG wire#powerrail
      Contact( "Station_Sys".Auto.AllRun )
   END_RUNG wire#w1
   // the same network as SCL:
   "ST10_FB_Tower_4Lamp_DB"(iReady := "Station_Sys".Status.Ready,   // "FB_Tower_4Lamp"
                           iManual_Mode := "Station_Sys".Manual.Mode,
                           iAuto_Mode := "Station_Sys".Auto.Mode,
                           iAuto_Running := "Station_Sys".Auto.Running OR "Station_Sys".Auto.AllRun,
                           iCheck_Mode := 0,
                           iIdle := 0,
                           iWarning := "Station_Sys".Warning.ON,
                           iFault := "Station_Sys".Alarm.ON,
                           "i0.5s_Pulse" := "ClockMemory0.5s",
                           i1s_Pulse := "ClockMemory1s",
                           i2s_Pulse := "ClockMemory2s",
                           iResetButton := "Station_Sys".Cmd.Reset,
                           "iE-StopButtonOK" := "Station_Sys".Status.EStopOK,
                           iSafetyGateClosed := "Station_Sys".Safety.DoorOK[0],
                           iSafetyGateRelayOK := "Station_Sys".Safety.DoorOK[0],
                           iPowerOn := "Station_Sys".Status.ControlOn,
                           iMachineHomePos := "Station_Sys".Initial.OK,
                           iWorkAreaLightButton := "ST10_GeneralData".HMI.StationLightPB,
                           iTest_Lamp := "Station_Sys".Cmd.TestLamp,
                           ioBuzzerON := "Station_Sys".Cmd.BuzzerOn,
                           oRed_Lamp => "oTowerLight-Red",
                           oYellow_Lamp => "oTowerLight-yellow",
                           oGreen_Lamp => "oTowerLight-Green",
                           oBlue_Lamp => "oTowerLight-Blue",
                           oBuzzer => "oTowerLight-Buzzer",
                           oPowerOn => "oHMIControlOn",
                           oResetLamp => "oHMIResetButton",
                           oWorkArea1_LightingOn => "oLED_lamp_1",
                           oWorkArea2_LightingOn => "oLED_lamp_2");
END_REGION

REGION Network 4: Q100.1 HMI启动按钮灯 / Q100.1 HMI Start button indicator
   RUNG wire#powerrail
      Contact( "Sys".COM.AlwaysON )
      wire#w1
      Contact( "Station_Sys".Initial.OK )
      Contact( "ClockMemory0.5s" )
      wire#w2
      Coil( "oHMIMachineStart" )
   END_RUNG
   RUNG wire#w1
      Contact( "Station_Sys".Cmd.TestLamp )
   END_RUNG wire#w2
   RUNG wire#w1
      Contact( "Station_Sys".Auto.AllRun )
   END_RUNG wire#w2
   // the same network as SCL:
   "oHMIMachineStart" := "Sys".COM.AlwaysON AND (("Station_Sys".Initial.OK AND "ClockMemory0.5s") OR "Station_Sys".Cmd.TestLamp OR "Station_Sys".Auto.AllRun);
END_REGION

REGION Network 5: Q100.2 HMI停止按钮灯 / Q100.2 HMI Stop button indicator
   RUNG wire#powerrail
      Contact( "Sys".COM.AlwaysON )
      wire#w1
      I_Contact( "Station_Sys".Initial.Running )
      I_Contact( "Station_Sys".Auto.AllRun )
      wire#w2
      Coil( "oHMIMachineStop" )
   END_RUNG
   RUNG wire#w1
      Contact( "Station_Sys".Cmd.TestLamp )
   END_RUNG wire#w2
   // the same network as SCL:
   "oHMIMachineStop" := "Sys".COM.AlwaysON AND ((NOT "Station_Sys".Initial.Running AND NOT "Station_Sys".Auto.AllRun) OR "Station_Sys".Cmd.TestLamp);
END_REGION

REGION Network 6: Q100.4 HMI开门按钮灯 / Q100.4 HMI Door opening button light
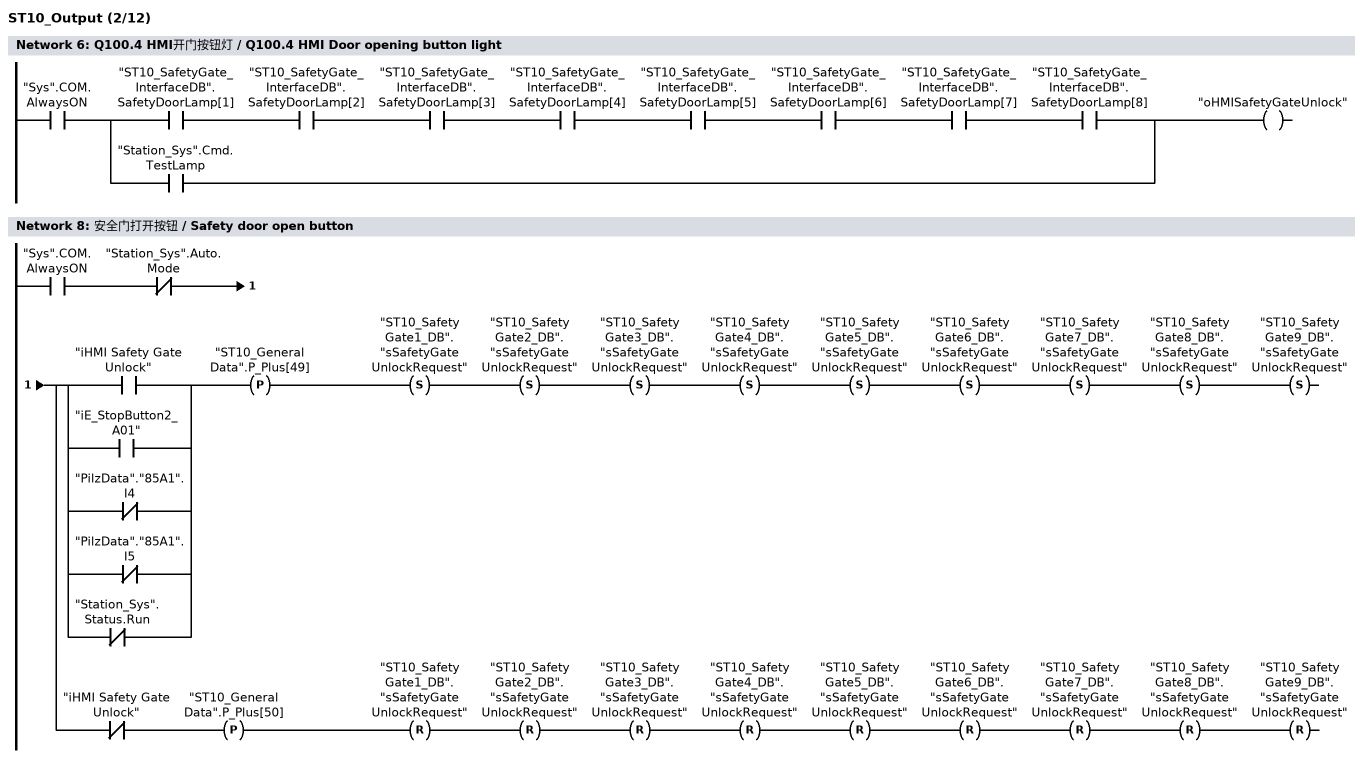
   RUNG wire#powerrail
      Contact( "Sys".COM.AlwaysON )
      wire#w1
      Contact( "ST10_SafetyGate_InterfaceDB".SafetyDoorLamp[1] )
      Contact( "ST10_SafetyGate_InterfaceDB".SafetyDoorLamp[2] )
      Contact( "ST10_SafetyGate_InterfaceDB".SafetyDoorLamp[3] )
      Contact( "ST10_SafetyGate_InterfaceDB".SafetyDoorLamp[4] )
      Contact( "ST10_SafetyGate_InterfaceDB".SafetyDoorLamp[5] )
      Contact( "ST10_SafetyGate_InterfaceDB".SafetyDoorLamp[6] )
      Contact( "ST10_SafetyGate_InterfaceDB".SafetyDoorLamp[7] )
      Contact( "ST10_SafetyGate_InterfaceDB".SafetyDoorLamp[8] )
      wire#w2
      Coil( "oHMISafetyGateUnlock" )
   END_RUNG
   RUNG wire#w1
      Contact( "Station_Sys".Cmd.TestLamp )
   END_RUNG wire#w2
   // the same network as SCL:
   "oHMISafetyGateUnlock" := "Sys".COM.AlwaysON AND (("ST10_SafetyGate_InterfaceDB".SafetyDoorLamp[1] AND "ST10_SafetyGate_InterfaceDB".SafetyDoorLamp[2] AND "ST10_SafetyGate_InterfaceDB".SafetyDoorLamp[3] AND "ST10_SafetyGate_InterfaceDB".SafetyDoorLamp[4] AND "ST10_SafetyGate_InterfaceDB".SafetyDoorLamp[5] AND "ST10_SafetyGate_InterfaceDB".SafetyDoorLamp[6] AND "ST10_SafetyGate_InterfaceDB".SafetyDoorLamp[7] AND "ST10_SafetyGate_InterfaceDB".SafetyDoorLamp[8]) OR "Station_Sys".Cmd.TestLamp);
END_REGION

REGION Network 8: 安全门打开按钮 / Safety door open button
   RUNG wire#powerrail
      Contact( "Sys".COM.AlwaysON )
      I_Contact( "Station_Sys".Auto.Mode )
      wire#w1
      Contact( "iHMI Safety Gate Unlock" )
      wire#w2
      P_Trig( "ST10_GeneralData".P_Plus[49] )
      S_Coil( "ST10_SafetyGate1_DB"."sSafetyGate UnlockRequest" )
      S_Coil( "ST10_SafetyGate2_DB"."sSafetyGate UnlockRequest" )
      S_Coil( "ST10_SafetyGate3_DB"."sSafetyGate UnlockRequest" )
      S_Coil( "ST10_SafetyGate4_DB"."sSafetyGate UnlockRequest" )
      S_Coil( "ST10_SafetyGate5_DB"."sSafetyGate UnlockRequest" )
      S_Coil( "ST10_SafetyGate6_DB"."sSafetyGate UnlockRequest" )
      S_Coil( "ST10_SafetyGate7_DB"."sSafetyGate UnlockRequest" )
      S_Coil( "ST10_SafetyGate8_DB"."sSafetyGate UnlockRequest" )
      S_Coil( "ST10_SafetyGate9_DB"."sSafetyGate UnlockRequest" )
   END_RUNG
   RUNG wire#w1
      Contact( "iE_StopButton2_A01" )
   END_RUNG wire#w2
   RUNG wire#w1
      I_Contact( "PilzData"."85A1".I4 )
   END_RUNG wire#w2
   RUNG wire#w1
      I_Contact( "PilzData"."85A1".I5 )
   END_RUNG wire#w2
   RUNG wire#w1
      I_Contact( "Station_Sys".Status.Run )
   END_RUNG wire#w2
   RUNG wire#w1
      I_Contact( "iHMI Safety Gate Unlock" )
      P_Trig( "ST10_GeneralData".P_Plus[50] )
      R_Coil( "ST10_SafetyGate1_DB"."sSafetyGate UnlockRequest" )
      R_Coil( "ST10_SafetyGate2_DB"."sSafetyGate UnlockRequest" )
      R_Coil( "ST10_SafetyGate3_DB"."sSafetyGate UnlockRequest" )
      R_Coil( "ST10_SafetyGate4_DB"."sSafetyGate UnlockRequest" )
      R_Coil( "ST10_SafetyGate5_DB"."sSafetyGate UnlockRequest" )
      R_Coil( "ST10_SafetyGate6_DB"."sSafetyGate UnlockRequest" )
      R_Coil( "ST10_SafetyGate7_DB"."sSafetyGate UnlockRequest" )
      R_Coil( "ST10_SafetyGate8_DB"."sSafetyGate UnlockRequest" )
      R_Coil( "ST10_SafetyGate9_DB"."sSafetyGate UnlockRequest" )
   END_RUNG
   // the same network as SCL:
   #_w1 := "Sys".COM.AlwaysON AND NOT "Station_Sys".Auto.Mode;
   #_w2 := #_w1 AND ("iHMI Safety Gate Unlock" OR "iE_StopButton2_A01" OR NOT "PilzData"."85A1".I4 OR NOT "PilzData"."85A1".I5 OR NOT "Station_Sys".Status.Run);
   #_w3 := #_w2 AND NOT "ST10_GeneralData".P_Plus[49];   // rising edge
   "ST10_GeneralData".P_Plus[49] := #_w2;
   IF #_w3 THEN
       "ST10_SafetyGate1_DB"."sSafetyGate UnlockRequest" := TRUE;
       "ST10_SafetyGate2_DB"."sSafetyGate UnlockRequest" := TRUE;
       "ST10_SafetyGate3_DB"."sSafetyGate UnlockRequest" := TRUE;
       "ST10_SafetyGate4_DB"."sSafetyGate UnlockRequest" := TRUE;
       "ST10_SafetyGate5_DB"."sSafetyGate UnlockRequest" := TRUE;
       "ST10_SafetyGate6_DB"."sSafetyGate UnlockRequest" := TRUE;
       "ST10_SafetyGate7_DB"."sSafetyGate UnlockRequest" := TRUE;
       "ST10_SafetyGate8_DB"."sSafetyGate UnlockRequest" := TRUE;
       "ST10_SafetyGate9_DB"."sSafetyGate UnlockRequest" := TRUE;
   END_IF;
   #_w4 := #_w1 AND NOT "iHMI Safety Gate Unlock";
   #_w5 := #_w4 AND NOT "ST10_GeneralData".P_Plus[50];   // rising edge
   "ST10_GeneralData".P_Plus[50] := #_w4;
   IF #_w5 THEN
       "ST10_SafetyGate1_DB"."sSafetyGate UnlockRequest" := FALSE;
       "ST10_SafetyGate2_DB"."sSafetyGate UnlockRequest" := FALSE;
       "ST10_SafetyGate3_DB"."sSafetyGate UnlockRequest" := FALSE;
       "ST10_SafetyGate4_DB"."sSafetyGate UnlockRequest" := FALSE;
       "ST10_SafetyGate5_DB"."sSafetyGate UnlockRequest" := FALSE;
       "ST10_SafetyGate6_DB"."sSafetyGate UnlockRequest" := FALSE;
       "ST10_SafetyGate7_DB"."sSafetyGate UnlockRequest" := FALSE;
       "ST10_SafetyGate8_DB"."sSafetyGate UnlockRequest" := FALSE;
       "ST10_SafetyGate9_DB"."sSafetyGate UnlockRequest" := FALSE;
   END_IF;
END_REGION

REGION Network 9: 安全门关闭 / Safety door closed
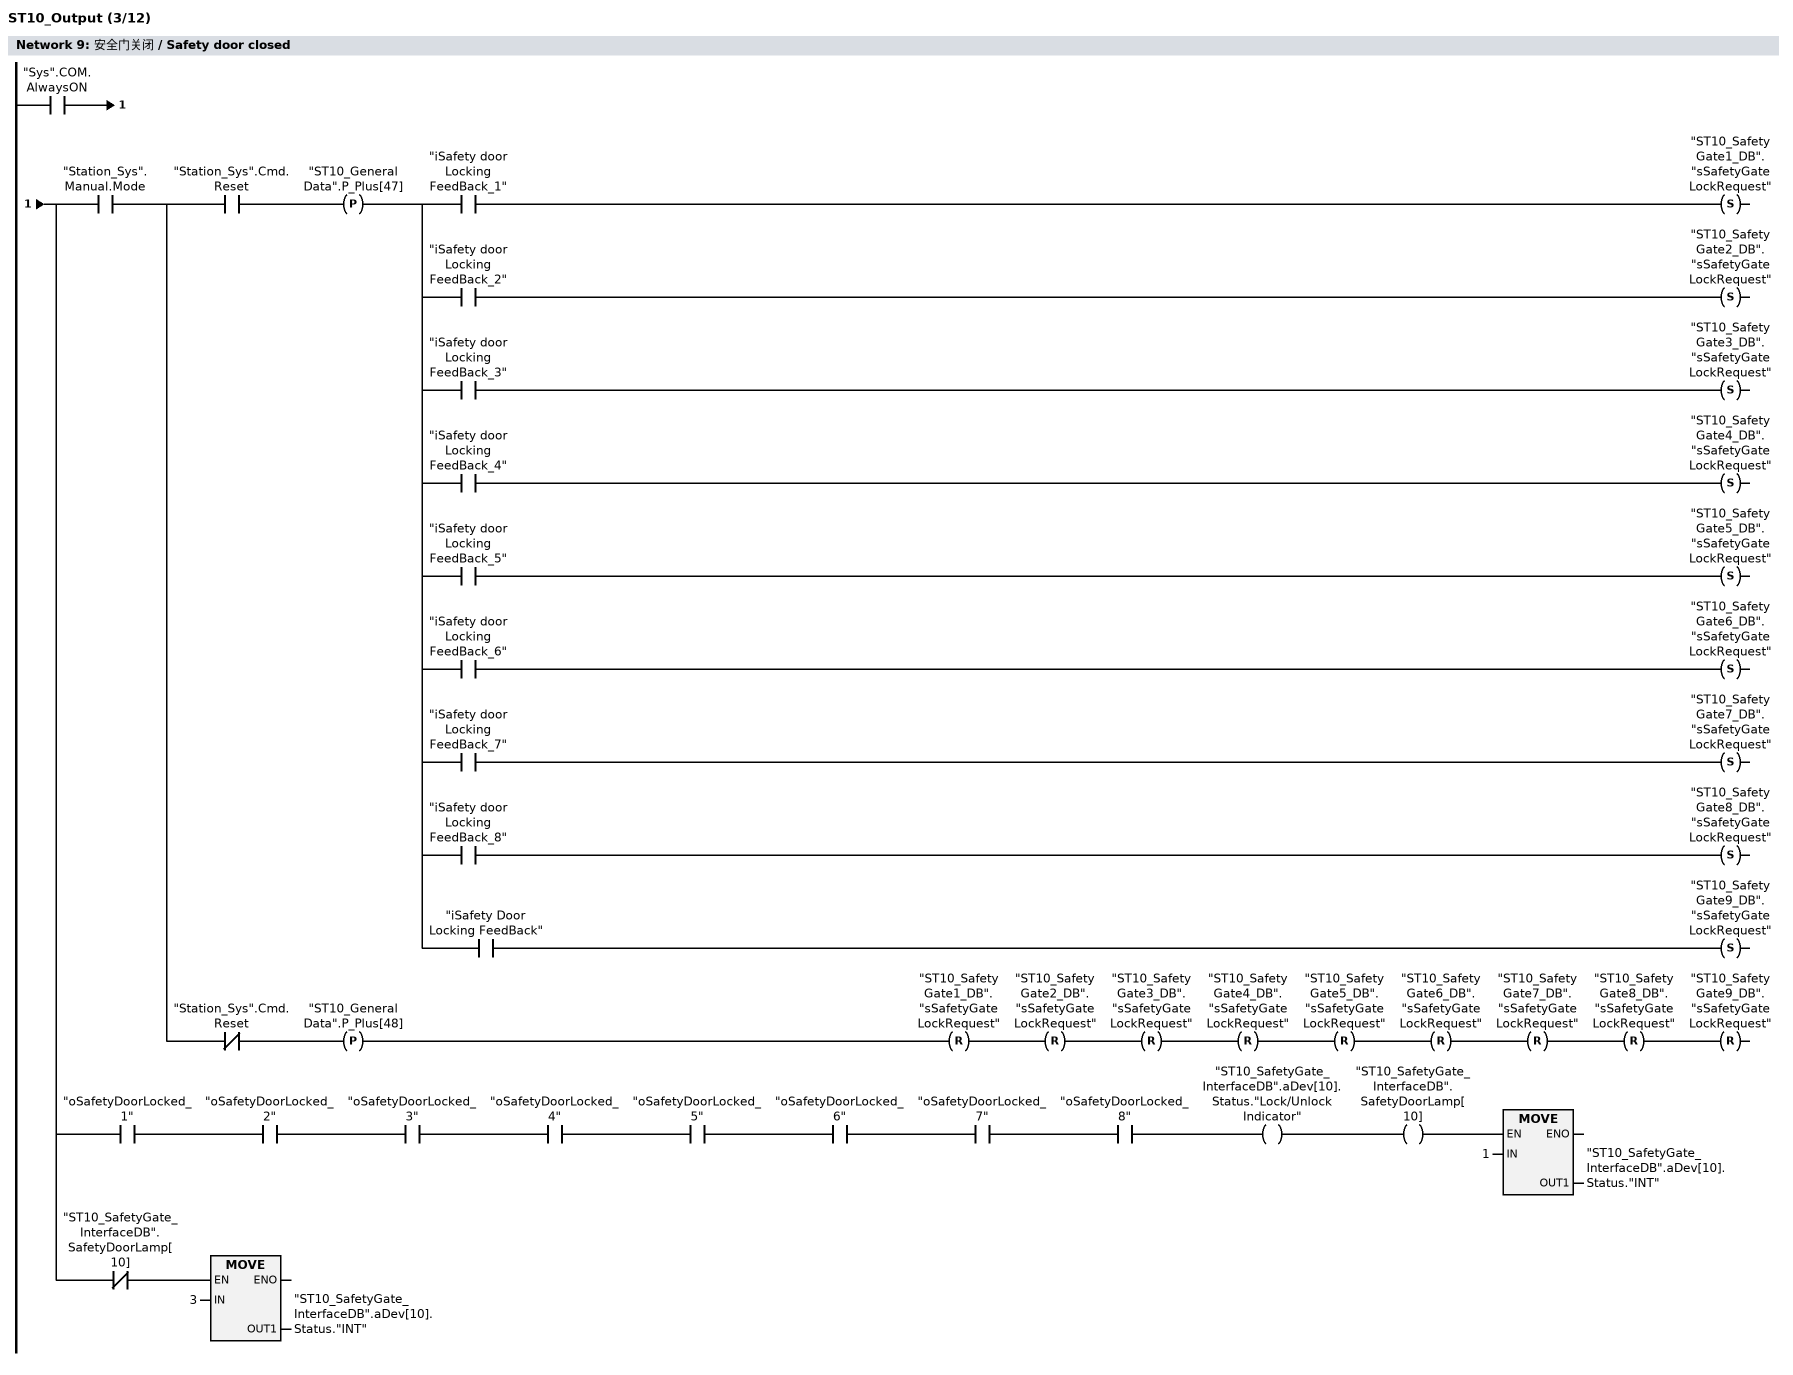
   RUNG wire#powerrail
      Contact( "Sys".COM.AlwaysON )
      wire#w1
      Contact( "Station_Sys".Manual.Mode )
      wire#w2
      Contact( "Station_Sys".Cmd.Reset )
      P_Trig( "ST10_GeneralData".P_Plus[47] )
      wire#w3
      Contact( "iSafety door Locking FeedBack_1" )
      S_Coil( "ST10_SafetyGate1_DB"."sSafetyGate LockRequest" )
   END_RUNG
   RUNG wire#w3
      Contact( "iSafety door Locking FeedBack_2" )
      S_Coil( "ST10_SafetyGate2_DB"."sSafetyGate LockRequest" )
   END_RUNG
   RUNG wire#w3
      Contact( "iSafety door Locking FeedBack_3" )
      S_Coil( "ST10_SafetyGate3_DB"."sSafetyGate LockRequest" )
   END_RUNG
   RUNG wire#w3
      Contact( "iSafety door Locking FeedBack_4" )
      S_Coil( "ST10_SafetyGate4_DB"."sSafetyGate LockRequest" )
   END_RUNG
   RUNG wire#w3
      Contact( "iSafety door Locking FeedBack_5" )
      S_Coil( "ST10_SafetyGate5_DB"."sSafetyGate LockRequest" )
   END_RUNG
   RUNG wire#w3
      Contact( "iSafety door Locking FeedBack_6" )
      S_Coil( "ST10_SafetyGate6_DB"."sSafetyGate LockRequest" )
   END_RUNG
   RUNG wire#w3
      Contact( "iSafety door Locking FeedBack_7" )
      S_Coil( "ST10_SafetyGate7_DB"."sSafetyGate LockRequest" )
   END_RUNG
   RUNG wire#w3
      Contact( "iSafety door Locking FeedBack_8" )
      S_Coil( "ST10_SafetyGate8_DB"."sSafetyGate LockRequest" )
   END_RUNG
   RUNG wire#w3
      Contact( "iSafety Door Locking FeedBack" )
      S_Coil( "ST10_SafetyGate9_DB"."sSafetyGate LockRequest" )
   END_RUNG
   RUNG wire#w2
      I_Contact( "Station_Sys".Cmd.Reset )
      P_Trig( "ST10_GeneralData".P_Plus[48] )
      R_Coil( "ST10_SafetyGate1_DB"."sSafetyGate LockRequest" )
      R_Coil( "ST10_SafetyGate2_DB"."sSafetyGate LockRequest" )
      R_Coil( "ST10_SafetyGate3_DB"."sSafetyGate LockRequest" )
      R_Coil( "ST10_SafetyGate4_DB"."sSafetyGate LockRequest" )
      R_Coil( "ST10_SafetyGate5_DB"."sSafetyGate LockRequest" )
      R_Coil( "ST10_SafetyGate6_DB"."sSafetyGate LockRequest" )
      R_Coil( "ST10_SafetyGate7_DB"."sSafetyGate LockRequest" )
      R_Coil( "ST10_SafetyGate8_DB"."sSafetyGate LockRequest" )
      R_Coil( "ST10_SafetyGate9_DB"."sSafetyGate LockRequest" )
   END_RUNG
   RUNG wire#w1
      Contact( "oSafetyDoorLocked_1" )
      Contact( "oSafetyDoorLocked_2" )
      Contact( "oSafetyDoorLocked_3" )
      Contact( "oSafetyDoorLocked_4" )
      Contact( "oSafetyDoorLocked_5" )
      Contact( "oSafetyDoorLocked_6" )
      Contact( "oSafetyDoorLocked_7" )
      Contact( "oSafetyDoorLocked_8" )
      Coil( "ST10_SafetyGate_InterfaceDB".aDev[10].Status."Lock/Unlock Indicator" )
      Coil( "ST10_SafetyGate_InterfaceDB".SafetyDoorLamp[10] )
      Move(in := 1, out1 => "ST10_SafetyGate_InterfaceDB".aDev[10].Status."INT")
   END_RUNG
   RUNG wire#w1
      I_Contact( "ST10_SafetyGate_InterfaceDB".SafetyDoorLamp[10] )
      Move(in := 3, out1 => "ST10_SafetyGate_InterfaceDB".aDev[10].Status."INT")
   END_RUNG
   // the same network as SCL:
   #_w1 := "Sys".COM.AlwaysON AND "Station_Sys".Manual.Mode;
   #_w2 := #_w1 AND "Station_Sys".Cmd.Reset;
   #_w3 := #_w2 AND NOT "ST10_GeneralData".P_Plus[47];   // rising edge
   "ST10_GeneralData".P_Plus[47] := #_w2;
   IF #_w3 AND "iSafety door Locking FeedBack_1" THEN
       "ST10_SafetyGate1_DB"."sSafetyGate LockRequest" := TRUE;
   END_IF;
   IF #_w3 AND "iSafety door Locking FeedBack_2" THEN
       "ST10_SafetyGate2_DB"."sSafetyGate LockRequest" := TRUE;
   END_IF;
   IF #_w3 AND "iSafety door Locking FeedBack_3" THEN
       "ST10_SafetyGate3_DB"."sSafetyGate LockRequest" := TRUE;
   END_IF;
   IF #_w3 AND "iSafety door Locking FeedBack_4" THEN
       "ST10_SafetyGate4_DB"."sSafetyGate LockRequest" := TRUE;
   END_IF;
   IF #_w3 AND "iSafety door Locking FeedBack_5" THEN
       "ST10_SafetyGate5_DB"."sSafetyGate LockRequest" := TRUE;
   END_IF;
   IF #_w3 AND "iSafety door Locking FeedBack_6" THEN
       "ST10_SafetyGate6_DB"."sSafetyGate LockRequest" := TRUE;
   END_IF;
   IF #_w3 AND "iSafety door Locking FeedBack_7" THEN
       "ST10_SafetyGate7_DB"."sSafetyGate LockRequest" := TRUE;
   END_IF;
   IF #_w3 AND "iSafety door Locking FeedBack_8" THEN
       "ST10_SafetyGate8_DB"."sSafetyGate LockRequest" := TRUE;
   END_IF;
   IF #_w3 AND "iSafety Door Locking FeedBack" THEN
       "ST10_SafetyGate9_DB"."sSafetyGate LockRequest" := TRUE;
   END_IF;
   #_w4 := #_w1 AND NOT "Station_Sys".Cmd.Reset;
   #_w5 := #_w4 AND NOT "ST10_GeneralData".P_Plus[48];   // rising edge
   "ST10_GeneralData".P_Plus[48] := #_w4;
   IF #_w5 THEN
       "ST10_SafetyGate1_DB"."sSafetyGate LockRequest" := FALSE;
       "ST10_SafetyGate2_DB"."sSafetyGate LockRequest" := FALSE;
       "ST10_SafetyGate3_DB"."sSafetyGate LockRequest" := FALSE;
       "ST10_SafetyGate4_DB"."sSafetyGate LockRequest" := FALSE;
       "ST10_SafetyGate5_DB"."sSafetyGate LockRequest" := FALSE;
       "ST10_SafetyGate6_DB"."sSafetyGate LockRequest" := FALSE;
       "ST10_SafetyGate7_DB"."sSafetyGate LockRequest" := FALSE;
       "ST10_SafetyGate8_DB"."sSafetyGate LockRequest" := FALSE;
       "ST10_SafetyGate9_DB"."sSafetyGate LockRequest" := FALSE;
   END_IF;
   "ST10_SafetyGate_InterfaceDB".aDev[10].Status."Lock/Unlock Indicator" := "Sys".COM.AlwaysON AND "oSafetyDoorLocked_1" AND "oSafetyDoorLocked_2" AND "oSafetyDoorLocked_3" AND "oSafetyDoorLocked_4" AND "oSafetyDoorLocked_5" AND "oSafetyDoorLocked_6" AND "oSafetyDoorLocked_7" AND "oSafetyDoorLocked_8";
   "ST10_SafetyGate_InterfaceDB".SafetyDoorLamp[10] := "Sys".COM.AlwaysON AND "oSafetyDoorLocked_1" AND "oSafetyDoorLocked_2" AND "oSafetyDoorLocked_3" AND "oSafetyDoorLocked_4" AND "oSafetyDoorLocked_5" AND "oSafetyDoorLocked_6" AND "oSafetyDoorLocked_7" AND "oSafetyDoorLocked_8";
   IF "Sys".COM.AlwaysON AND "oSafetyDoorLocked_1" AND "oSafetyDoorLocked_2" AND "oSafetyDoorLocked_3" AND "oSafetyDoorLocked_4" AND "oSafetyDoorLocked_5" AND "oSafetyDoorLocked_6" AND "oSafetyDoorLocked_7" AND "oSafetyDoorLocked_8" THEN
       "ST10_SafetyGate_InterfaceDB".aDev[10].Status."INT" := 1;
   END_IF;
   IF "Sys".COM.AlwaysON AND NOT "ST10_SafetyGate_InterfaceDB".SafetyDoorLamp[10] THEN
       "ST10_SafetyGate_InterfaceDB".aDev[10].Status."INT" := 3;
   END_IF;
END_REGION

REGION Network 11: E-NG料盒-01安全门锁按钮灯 / E-NG Material Box -01 Security door lock button light
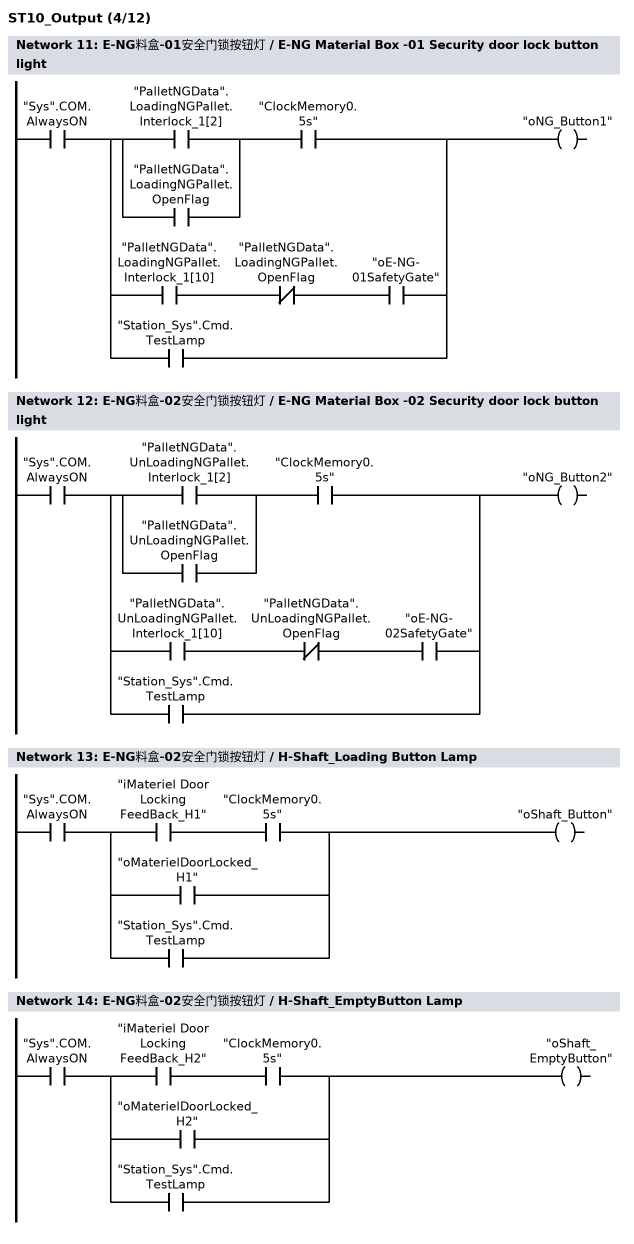
   RUNG wire#powerrail
      Contact( "Sys".COM.AlwaysON )
      wire#w1
      Contact( "PalletNGData".LoadingNGPallet.Interlock_1[2] )
      wire#w2
      Contact( "ClockMemory0.5s" )
      wire#w3
      Coil( "oNG_Button1" )
   END_RUNG
   RUNG wire#w1
      Contact( "PalletNGData".LoadingNGPallet.OpenFlag )
   END_RUNG wire#w2
   RUNG wire#w1
      Contact( "PalletNGData".LoadingNGPallet.Interlock_1[10] )
      I_Contact( "PalletNGData".LoadingNGPallet.OpenFlag )
      Contact( "oE-NG-01SafetyGate" )
   END_RUNG wire#w3
   RUNG wire#w1
      Contact( "Station_Sys".Cmd.TestLamp )
   END_RUNG wire#w3
   // the same network as SCL:
   "oNG_Button1" := "Sys".COM.AlwaysON AND ((("PalletNGData".LoadingNGPallet.Interlock_1[2] OR "PalletNGData".LoadingNGPallet.OpenFlag) AND "ClockMemory0.5s") OR ("PalletNGData".LoadingNGPallet.Interlock_1[10] AND NOT "PalletNGData".LoadingNGPallet.OpenFlag AND "oE-NG-01SafetyGate") OR "Station_Sys".Cmd.TestLamp);
END_REGION

REGION Network 12: E-NG料盒-02安全门锁按钮灯 / E-NG Material Box -02 Security door lock button light
   RUNG wire#powerrail
      Contact( "Sys".COM.AlwaysON )
      wire#w1
      Contact( "PalletNGData".UnLoadingNGPallet.Interlock_1[2] )
      wire#w2
      Contact( "ClockMemory0.5s" )
      wire#w3
      Coil( "oNG_Button2" )
   END_RUNG
   RUNG wire#w1
      Contact( "PalletNGData".UnLoadingNGPallet.OpenFlag )
   END_RUNG wire#w2
   RUNG wire#w1
      Contact( "PalletNGData".UnLoadingNGPallet.Interlock_1[10] )
      I_Contact( "PalletNGData".UnLoadingNGPallet.OpenFlag )
      Contact( "oE-NG-02SafetyGate" )
   END_RUNG wire#w3
   RUNG wire#w1
      Contact( "Station_Sys".Cmd.TestLamp )
   END_RUNG wire#w3
   // the same network as SCL:
   "oNG_Button2" := "Sys".COM.AlwaysON AND ((("PalletNGData".UnLoadingNGPallet.Interlock_1[2] OR "PalletNGData".UnLoadingNGPallet.OpenFlag) AND "ClockMemory0.5s") OR ("PalletNGData".UnLoadingNGPallet.Interlock_1[10] AND NOT "PalletNGData".UnLoadingNGPallet.OpenFlag AND "oE-NG-02SafetyGate") OR "Station_Sys".Cmd.TestLamp);
END_REGION

REGION Network 13: E-NG料盒-02安全门锁按钮灯 / H-Shaft_Loading Button Lamp
   RUNG wire#powerrail
      Contact( "Sys".COM.AlwaysON )
      wire#w1
      Contact( "iMateriel Door Locking FeedBack_H1" )
      Contact( "ClockMemory0.5s" )
      wire#w2
      Coil( "oShaft_Button" )
   END_RUNG
   RUNG wire#w1
      Contact( "oMaterielDoorLocked_H1" )
   END_RUNG wire#w2
   RUNG wire#w1
      Contact( "Station_Sys".Cmd.TestLamp )
   END_RUNG wire#w2
   // the same network as SCL:
   "oShaft_Button" := "Sys".COM.AlwaysON AND (("iMateriel Door Locking FeedBack_H1" AND "ClockMemory0.5s") OR "oMaterielDoorLocked_H1" OR "Station_Sys".Cmd.TestLamp);
END_REGION

REGION Network 14: E-NG料盒-02安全门锁按钮灯 / H-Shaft_EmptyButton Lamp
   RUNG wire#powerrail
      Contact( "Sys".COM.AlwaysON )
      wire#w1
      Contact( "iMateriel Door Locking FeedBack_H2" )
      Contact( "ClockMemory0.5s" )
      wire#w2
      Coil( "oShaft_EmptyButton" )
   END_RUNG
   RUNG wire#w1
      Contact( "oMaterielDoorLocked_H2" )
   END_RUNG wire#w2
   RUNG wire#w1
      Contact( "Station_Sys".Cmd.TestLamp )
   END_RUNG wire#w2
   // the same network as SCL:
   "oShaft_EmptyButton" := "Sys".COM.AlwaysON AND (("iMateriel Door Locking FeedBack_H2" AND "ClockMemory0.5s") OR "oMaterielDoorLocked_H2" OR "Station_Sys".Cmd.TestLamp);
END_REGION

REGION Network 15: E-NG料盒-02安全门锁按钮灯 / H-Shaft_Loading DoorButton Lamp 6
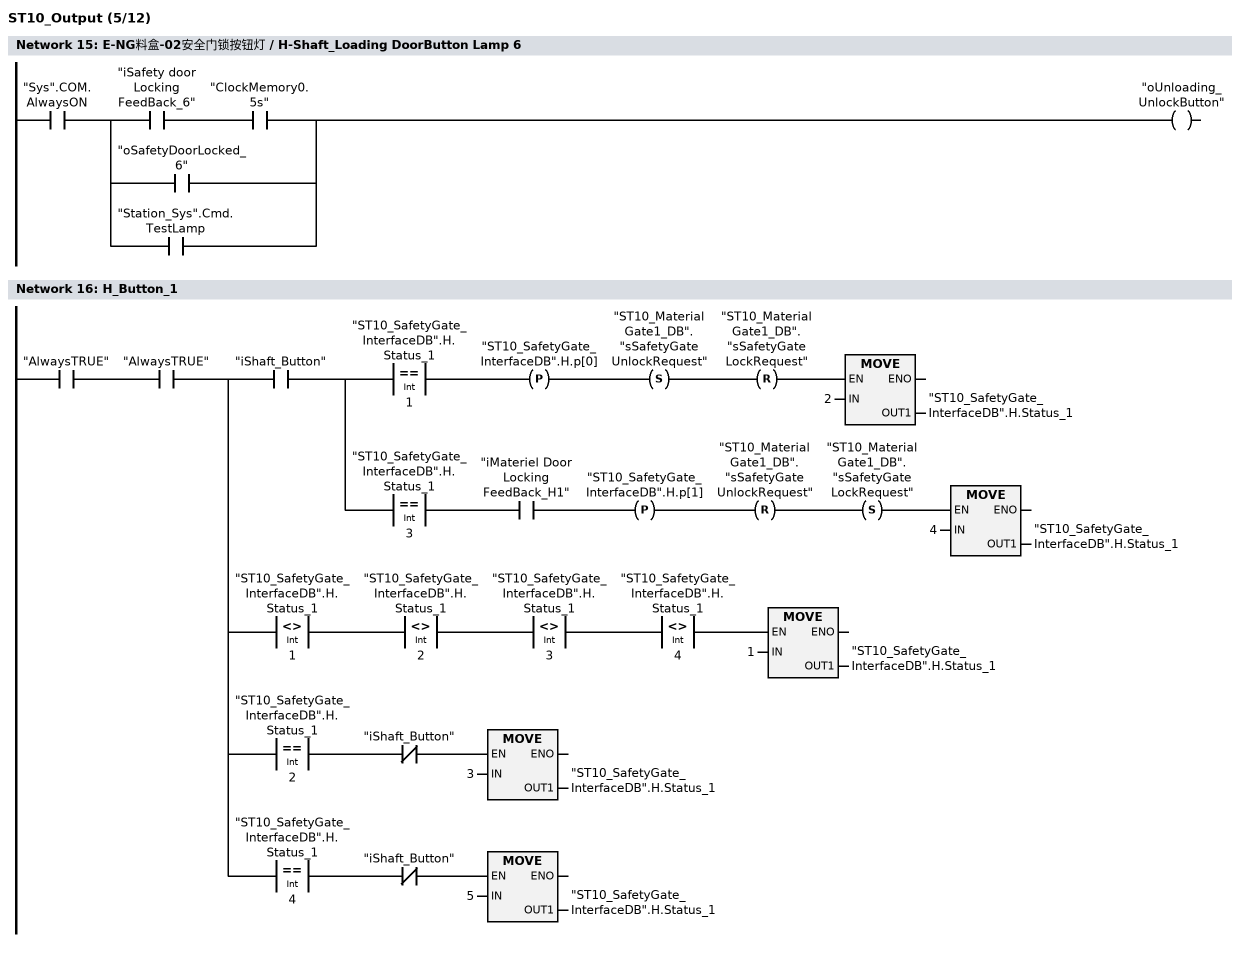
   RUNG wire#powerrail
      Contact( "Sys".COM.AlwaysON )
      wire#w1
      Contact( "iSafety door Locking FeedBack_6" )
      Contact( "ClockMemory0.5s" )
      wire#w2
      Coil( "oUnloading_UnlockButton" )
   END_RUNG
   RUNG wire#w1
      Contact( "oSafetyDoorLocked_6" )
   END_RUNG wire#w2
   RUNG wire#w1
      Contact( "Station_Sys".Cmd.TestLamp )
   END_RUNG wire#w2
   // the same network as SCL:
   "oUnloading_UnlockButton" := "Sys".COM.AlwaysON AND (("iSafety door Locking FeedBack_6" AND "ClockMemory0.5s") OR "oSafetyDoorLocked_6" OR "Station_Sys".Cmd.TestLamp);
END_REGION

REGION Network 16: H_Button_1
   RUNG wire#powerrail
      Contact( "AlwaysTRUE" )
      Contact( "AlwaysTRUE" )
      wire#w1
      Contact( "iShaft_Button" )
      wire#w2
      { S7_Templates := "SrcType := Int" } EQ_Contact(in1 := "ST10_SafetyGate_InterfaceDB".H.Status_1, in2 := 1)
      P_Trig( "ST10_SafetyGate_InterfaceDB".H.p[0] )
      S_Coil( "ST10_MaterialGate1_DB"."sSafetyGate UnlockRequest" )
      R_Coil( "ST10_MaterialGate1_DB"."sSafetyGate LockRequest" )
      Move(in := 2, out1 => "ST10_SafetyGate_InterfaceDB".H.Status_1)
   END_RUNG
   RUNG wire#w2
      { S7_Templates := "SrcType := Int" } EQ_Contact(in1 := "ST10_SafetyGate_InterfaceDB".H.Status_1, in2 := 3)
      Contact( "iMateriel Door Locking FeedBack_H1" )
      P_Trig( "ST10_SafetyGate_InterfaceDB".H.p[1] )
      R_Coil( "ST10_MaterialGate1_DB"."sSafetyGate UnlockRequest" )
      S_Coil( "ST10_MaterialGate1_DB"."sSafetyGate LockRequest" )
      Move(in := 4, out1 => "ST10_SafetyGate_InterfaceDB".H.Status_1)
   END_RUNG
   RUNG wire#w1
      { S7_Templates := "SrcType := Int" } NE_Contact(in1 := "ST10_SafetyGate_InterfaceDB".H.Status_1, in2 := 1)
      { S7_Templates := "SrcType := Int" } NE_Contact(in1 := "ST10_SafetyGate_InterfaceDB".H.Status_1, in2 := 2)
      { S7_Templates := "SrcType := Int" } NE_Contact(in1 := "ST10_SafetyGate_InterfaceDB".H.Status_1, in2 := 3)
      { S7_Templates := "SrcType := Int" } NE_Contact(in1 := "ST10_SafetyGate_InterfaceDB".H.Status_1, in2 := 4)
      Move(in := 1, out1 => "ST10_SafetyGate_InterfaceDB".H.Status_1)
   END_RUNG
   RUNG wire#w1
      { S7_Templates := "SrcType := Int" } EQ_Contact(in1 := "ST10_SafetyGate_InterfaceDB".H.Status_1, in2 := 2)
      I_Contact( "iShaft_Button" )
      Move(in := 3, out1 => "ST10_SafetyGate_InterfaceDB".H.Status_1)
   END_RUNG
   RUNG wire#w1
      { S7_Templates := "SrcType := Int" } EQ_Contact(in1 := "ST10_SafetyGate_InterfaceDB".H.Status_1, in2 := 4)
      I_Contact( "iShaft_Button" )
      Move(in := 5, out1 => "ST10_SafetyGate_InterfaceDB".H.Status_1)
   END_RUNG
   // the same network as SCL:
   #_w1 := "AlwaysTRUE" AND "AlwaysTRUE";
   #_w2 := #_w1 AND "iShaft_Button";
   #_w3 := #_w2 AND ("ST10_SafetyGate_InterfaceDB".H.Status_1 = 1);
   #_w4 := #_w3 AND NOT "ST10_SafetyGate_InterfaceDB".H.p[0];   // rising edge
   "ST10_SafetyGate_InterfaceDB".H.p[0] := #_w3;
   IF #_w4 THEN
       "ST10_MaterialGate1_DB"."sSafetyGate UnlockRequest" := TRUE;
       "ST10_MaterialGate1_DB"."sSafetyGate LockRequest" := FALSE;
       "ST10_SafetyGate_InterfaceDB".H.Status_1 := 2;
   END_IF;
   #_w5 := #_w2 AND ("ST10_SafetyGate_InterfaceDB".H.Status_1 = 3) AND "iMateriel Door Locking FeedBack_H1";
   #_w6 := #_w5 AND NOT "ST10_SafetyGate_InterfaceDB".H.p[1];   // rising edge
   "ST10_SafetyGate_InterfaceDB".H.p[1] := #_w5;
   IF #_w6 THEN
       "ST10_MaterialGate1_DB"."sSafetyGate UnlockRequest" := FALSE;
       "ST10_MaterialGate1_DB"."sSafetyGate LockRequest" := TRUE;
       "ST10_SafetyGate_InterfaceDB".H.Status_1 := 4;
   END_IF;
   IF #_w1 AND ("ST10_SafetyGate_InterfaceDB".H.Status_1 <> 1) AND ("ST10_SafetyGate_InterfaceDB".H.Status_1 <> 2) AND ("ST10_SafetyGate_InterfaceDB".H.Status_1 <> 3) AND ("ST10_SafetyGate_InterfaceDB".H.Status_1 <> 4) THEN
       "ST10_SafetyGate_InterfaceDB".H.Status_1 := 1;
   END_IF;
   IF #_w1 AND ("ST10_SafetyGate_InterfaceDB".H.Status_1 = 2) AND NOT "iShaft_Button" THEN
       "ST10_SafetyGate_InterfaceDB".H.Status_1 := 3;
   END_IF;
   IF #_w1 AND ("ST10_SafetyGate_InterfaceDB".H.Status_1 = 4) AND NOT "iShaft_Button" THEN
       "ST10_SafetyGate_InterfaceDB".H.Status_1 := 5;
   END_IF;
END_REGION

REGION Network 17: H_Button_2
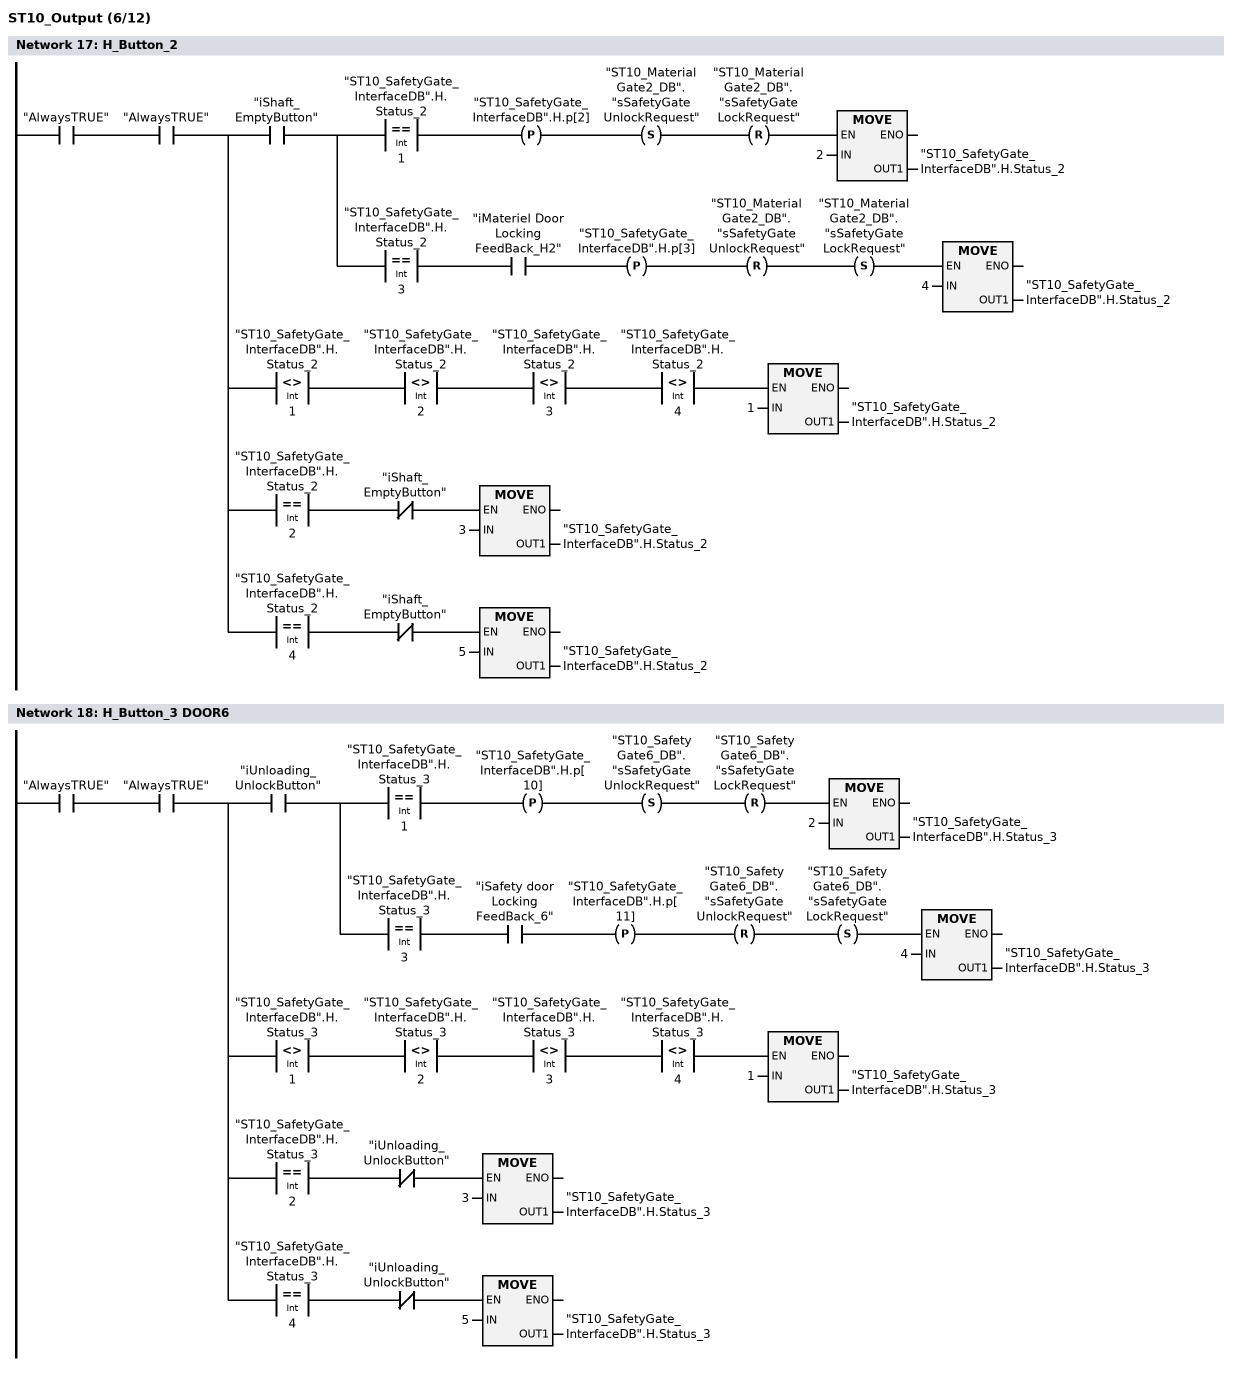
   RUNG wire#powerrail
      Contact( "AlwaysTRUE" )
      Contact( "AlwaysTRUE" )
      wire#w1
      Contact( "iShaft_EmptyButton" )
      wire#w2
      { S7_Templates := "SrcType := Int" } EQ_Contact(in1 := "ST10_SafetyGate_InterfaceDB".H.Status_2, in2 := 1)
      P_Trig( "ST10_SafetyGate_InterfaceDB".H.p[2] )
      S_Coil( "ST10_MaterialGate2_DB"."sSafetyGate UnlockRequest" )
      R_Coil( "ST10_MaterialGate2_DB"."sSafetyGate LockRequest" )
      Move(in := 2, out1 => "ST10_SafetyGate_InterfaceDB".H.Status_2)
   END_RUNG
   RUNG wire#w2
      { S7_Templates := "SrcType := Int" } EQ_Contact(in1 := "ST10_SafetyGate_InterfaceDB".H.Status_2, in2 := 3)
      Contact( "iMateriel Door Locking FeedBack_H2" )
      P_Trig( "ST10_SafetyGate_InterfaceDB".H.p[3] )
      R_Coil( "ST10_MaterialGate2_DB"."sSafetyGate UnlockRequest" )
      S_Coil( "ST10_MaterialGate2_DB"."sSafetyGate LockRequest" )
      Move(in := 4, out1 => "ST10_SafetyGate_InterfaceDB".H.Status_2)
   END_RUNG
   RUNG wire#w1
      { S7_Templates := "SrcType := Int" } NE_Contact(in1 := "ST10_SafetyGate_InterfaceDB".H.Status_2, in2 := 1)
      { S7_Templates := "SrcType := Int" } NE_Contact(in1 := "ST10_SafetyGate_InterfaceDB".H.Status_2, in2 := 2)
      { S7_Templates := "SrcType := Int" } NE_Contact(in1 := "ST10_SafetyGate_InterfaceDB".H.Status_2, in2 := 3)
      { S7_Templates := "SrcType := Int" } NE_Contact(in1 := "ST10_SafetyGate_InterfaceDB".H.Status_2, in2 := 4)
      Move(in := 1, out1 => "ST10_SafetyGate_InterfaceDB".H.Status_2)
   END_RUNG
   RUNG wire#w1
      { S7_Templates := "SrcType := Int" } EQ_Contact(in1 := "ST10_SafetyGate_InterfaceDB".H.Status_2, in2 := 2)
      I_Contact( "iShaft_EmptyButton" )
      Move(in := 3, out1 => "ST10_SafetyGate_InterfaceDB".H.Status_2)
   END_RUNG
   RUNG wire#w1
      { S7_Templates := "SrcType := Int" } EQ_Contact(in1 := "ST10_SafetyGate_InterfaceDB".H.Status_2, in2 := 4)
      I_Contact( "iShaft_EmptyButton" )
      Move(in := 5, out1 => "ST10_SafetyGate_InterfaceDB".H.Status_2)
   END_RUNG
   // the same network as SCL:
   #_w1 := "AlwaysTRUE" AND "AlwaysTRUE";
   #_w2 := #_w1 AND "iShaft_EmptyButton";
   #_w3 := #_w2 AND ("ST10_SafetyGate_InterfaceDB".H.Status_2 = 1);
   #_w4 := #_w3 AND NOT "ST10_SafetyGate_InterfaceDB".H.p[2];   // rising edge
   "ST10_SafetyGate_InterfaceDB".H.p[2] := #_w3;
   IF #_w4 THEN
       "ST10_MaterialGate2_DB"."sSafetyGate UnlockRequest" := TRUE;
       "ST10_MaterialGate2_DB"."sSafetyGate LockRequest" := FALSE;
       "ST10_SafetyGate_InterfaceDB".H.Status_2 := 2;
   END_IF;
   #_w5 := #_w2 AND ("ST10_SafetyGate_InterfaceDB".H.Status_2 = 3) AND "iMateriel Door Locking FeedBack_H2";
   #_w6 := #_w5 AND NOT "ST10_SafetyGate_InterfaceDB".H.p[3];   // rising edge
   "ST10_SafetyGate_InterfaceDB".H.p[3] := #_w5;
   IF #_w6 THEN
       "ST10_MaterialGate2_DB"."sSafetyGate UnlockRequest" := FALSE;
       "ST10_MaterialGate2_DB"."sSafetyGate LockRequest" := TRUE;
       "ST10_SafetyGate_InterfaceDB".H.Status_2 := 4;
   END_IF;
   IF #_w1 AND ("ST10_SafetyGate_InterfaceDB".H.Status_2 <> 1) AND ("ST10_SafetyGate_InterfaceDB".H.Status_2 <> 2) AND ("ST10_SafetyGate_InterfaceDB".H.Status_2 <> 3) AND ("ST10_SafetyGate_InterfaceDB".H.Status_2 <> 4) THEN
       "ST10_SafetyGate_InterfaceDB".H.Status_2 := 1;
   END_IF;
   IF #_w1 AND ("ST10_SafetyGate_InterfaceDB".H.Status_2 = 2) AND NOT "iShaft_EmptyButton" THEN
       "ST10_SafetyGate_InterfaceDB".H.Status_2 := 3;
   END_IF;
   IF #_w1 AND ("ST10_SafetyGate_InterfaceDB".H.Status_2 = 4) AND NOT "iShaft_EmptyButton" THEN
       "ST10_SafetyGate_InterfaceDB".H.Status_2 := 5;
   END_IF;
END_REGION

REGION Network 18: H_Button_3 DOOR6
   RUNG wire#powerrail
      Contact( "AlwaysTRUE" )
      Contact( "AlwaysTRUE" )
      wire#w1
      Contact( "iUnloading_UnlockButton" )
      wire#w2
      { S7_Templates := "SrcType := Int" } EQ_Contact(in1 := "ST10_SafetyGate_InterfaceDB".H.Status_3, in2 := 1)
      P_Trig( "ST10_SafetyGate_InterfaceDB".H.p[10] )
      S_Coil( "ST10_SafetyGate6_DB"."sSafetyGate UnlockRequest" )
      R_Coil( "ST10_SafetyGate6_DB"."sSafetyGate LockRequest" )
      Move(in := 2, out1 => "ST10_SafetyGate_InterfaceDB".H.Status_3)
   END_RUNG
   RUNG wire#w2
      { S7_Templates := "SrcType := Int" } EQ_Contact(in1 := "ST10_SafetyGate_InterfaceDB".H.Status_3, in2 := 3)
      Contact( "iSafety door Locking FeedBack_6" )
      P_Trig( "ST10_SafetyGate_InterfaceDB".H.p[11] )
      R_Coil( "ST10_SafetyGate6_DB"."sSafetyGate UnlockRequest" )
      S_Coil( "ST10_SafetyGate6_DB"."sSafetyGate LockRequest" )
      Move(in := 4, out1 => "ST10_SafetyGate_InterfaceDB".H.Status_3)
   END_RUNG
   RUNG wire#w1
      { S7_Templates := "SrcType := Int" } NE_Contact(in1 := "ST10_SafetyGate_InterfaceDB".H.Status_3, in2 := 1)
      { S7_Templates := "SrcType := Int" } NE_Contact(in1 := "ST10_SafetyGate_InterfaceDB".H.Status_3, in2 := 2)
      { S7_Templates := "SrcType := Int" } NE_Contact(in1 := "ST10_SafetyGate_InterfaceDB".H.Status_3, in2 := 3)
      { S7_Templates := "SrcType := Int" } NE_Contact(in1 := "ST10_SafetyGate_InterfaceDB".H.Status_3, in2 := 4)
      Move(in := 1, out1 => "ST10_SafetyGate_InterfaceDB".H.Status_3)
   END_RUNG
   RUNG wire#w1
      { S7_Templates := "SrcType := Int" } EQ_Contact(in1 := "ST10_SafetyGate_InterfaceDB".H.Status_3, in2 := 2)
      I_Contact( "iUnloading_UnlockButton" )
      Move(in := 3, out1 => "ST10_SafetyGate_InterfaceDB".H.Status_3)
   END_RUNG
   RUNG wire#w1
      { S7_Templates := "SrcType := Int" } EQ_Contact(in1 := "ST10_SafetyGate_InterfaceDB".H.Status_3, in2 := 4)
      I_Contact( "iUnloading_UnlockButton" )
      Move(in := 5, out1 => "ST10_SafetyGate_InterfaceDB".H.Status_3)
   END_RUNG
   // the same network as SCL:
   #_w1 := "AlwaysTRUE" AND "AlwaysTRUE";
   #_w2 := #_w1 AND "iUnloading_UnlockButton";
   #_w3 := #_w2 AND ("ST10_SafetyGate_InterfaceDB".H.Status_3 = 1);
   #_w4 := #_w3 AND NOT "ST10_SafetyGate_InterfaceDB".H.p[10];   // rising edge
   "ST10_SafetyGate_InterfaceDB".H.p[10] := #_w3;
   IF #_w4 THEN
       "ST10_SafetyGate6_DB"."sSafetyGate UnlockRequest" := TRUE;
       "ST10_SafetyGate6_DB"."sSafetyGate LockRequest" := FALSE;
       "ST10_SafetyGate_InterfaceDB".H.Status_3 := 2;
   END_IF;
   #_w5 := #_w2 AND ("ST10_SafetyGate_InterfaceDB".H.Status_3 = 3) AND "iSafety door Locking FeedBack_6";
   #_w6 := #_w5 AND NOT "ST10_SafetyGate_InterfaceDB".H.p[11];   // rising edge
   "ST10_SafetyGate_InterfaceDB".H.p[11] := #_w5;
   IF #_w6 THEN
       "ST10_SafetyGate6_DB"."sSafetyGate UnlockRequest" := FALSE;
       "ST10_SafetyGate6_DB"."sSafetyGate LockRequest" := TRUE;
       "ST10_SafetyGate_InterfaceDB".H.Status_3 := 4;
   END_IF;
   IF #_w1 AND ("ST10_SafetyGate_InterfaceDB".H.Status_3 <> 1) AND ("ST10_SafetyGate_InterfaceDB".H.Status_3 <> 2) AND ("ST10_SafetyGate_InterfaceDB".H.Status_3 <> 3) AND ("ST10_SafetyGate_InterfaceDB".H.Status_3 <> 4) THEN
       "ST10_SafetyGate_InterfaceDB".H.Status_3 := 1;
   END_IF;
   IF #_w1 AND ("ST10_SafetyGate_InterfaceDB".H.Status_3 = 2) AND NOT "iUnloading_UnlockButton" THEN
       "ST10_SafetyGate_InterfaceDB".H.Status_3 := 3;
   END_IF;
   IF #_w1 AND ("ST10_SafetyGate_InterfaceDB".H.Status_3 = 4) AND NOT "iUnloading_UnlockButton" THEN
       "ST10_SafetyGate_InterfaceDB".H.Status_3 := 5;
   END_IF;
END_REGION

REGION Network 19: E-NG料盒-02安全门锁按钮灯 / J-Magnet_Loading Button Lamp
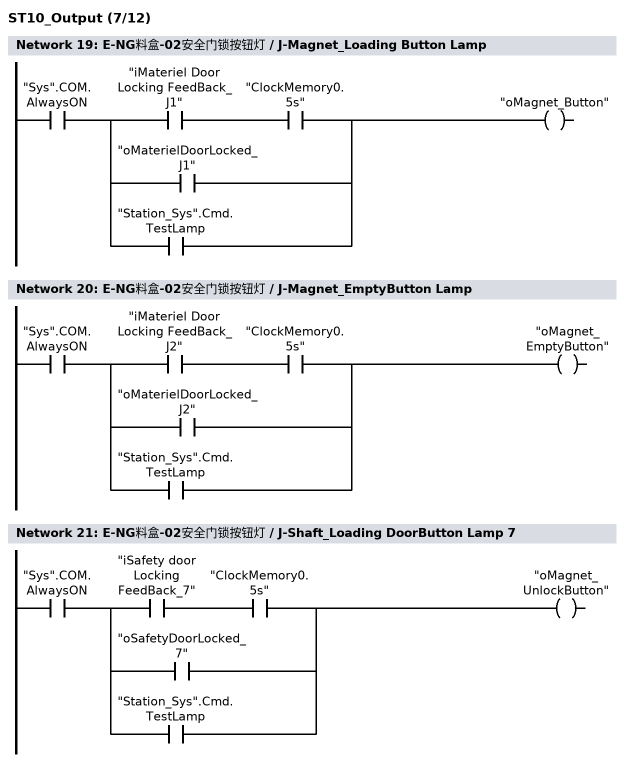
   RUNG wire#powerrail
      Contact( "Sys".COM.AlwaysON )
      wire#w1
      Contact( "iMateriel Door Locking FeedBack_J1" )
      Contact( "ClockMemory0.5s" )
      wire#w2
      Coil( "oMagnet_Button" )
   END_RUNG
   RUNG wire#w1
      Contact( "oMaterielDoorLocked_J1" )
   END_RUNG wire#w2
   RUNG wire#w1
      Contact( "Station_Sys".Cmd.TestLamp )
   END_RUNG wire#w2
   // the same network as SCL:
   "oMagnet_Button" := "Sys".COM.AlwaysON AND (("iMateriel Door Locking FeedBack_J1" AND "ClockMemory0.5s") OR "oMaterielDoorLocked_J1" OR "Station_Sys".Cmd.TestLamp);
END_REGION

REGION Network 20: E-NG料盒-02安全门锁按钮灯 / J-Magnet_EmptyButton Lamp
   RUNG wire#powerrail
      Contact( "Sys".COM.AlwaysON )
      wire#w1
      Contact( "iMateriel Door Locking FeedBack_J2" )
      Contact( "ClockMemory0.5s" )
      wire#w2
      Coil( "oMagnet_EmptyButton" )
   END_RUNG
   RUNG wire#w1
      Contact( "oMaterielDoorLocked_J2" )
   END_RUNG wire#w2
   RUNG wire#w1
      Contact( "Station_Sys".Cmd.TestLamp )
   END_RUNG wire#w2
   // the same network as SCL:
   "oMagnet_EmptyButton" := "Sys".COM.AlwaysON AND (("iMateriel Door Locking FeedBack_J2" AND "ClockMemory0.5s") OR "oMaterielDoorLocked_J2" OR "Station_Sys".Cmd.TestLamp);
END_REGION

REGION Network 21: E-NG料盒-02安全门锁按钮灯 / J-Shaft_Loading DoorButton Lamp 7
   RUNG wire#powerrail
      Contact( "Sys".COM.AlwaysON )
      wire#w1
      Contact( "iSafety door Locking FeedBack_7" )
      Contact( "ClockMemory0.5s" )
      wire#w2
      Coil( "oMagnet_UnlockButton" )
   END_RUNG
   RUNG wire#w1
      Contact( "oSafetyDoorLocked_7" )
   END_RUNG wire#w2
   RUNG wire#w1
      Contact( "Station_Sys".Cmd.TestLamp )
   END_RUNG wire#w2
   // the same network as SCL:
   "oMagnet_UnlockButton" := "Sys".COM.AlwaysON AND (("iSafety door Locking FeedBack_7" AND "ClockMemory0.5s") OR "oSafetyDoorLocked_7" OR "Station_Sys".Cmd.TestLamp);
END_REGION

